// TIA Portal V20 export
// export: Created 2025-12-01T14:56:34.8716322Z, ExportSetting None, DisplayName Totally Integrated Automation Portal, DisplayVersion V20 Update 3, DisplayName TIA Portal Openness, DisplayVersion V20 Update 3, DisplayName TIA Portal Version Control Interface, DisplayVersion V20 Update 3, DisplayName STEP 7 Professional, DisplayVersion V20 Update 3, DisplayName STEP 7 Safety, DisplayVersion V20 Update 2, DisplayName WinCC Basic/Comfort/Advanced, DisplayVersion V20 Update 3, DisplayName WinCC Professional, DisplayVersion V20 Update 3, DisplayName WinCC Unified, DisplayVersion V20 Update 3
FUNCTION_BLOCK "FB464_CRTL_TR_TP_E124_S34_Pres"   // FB464, LAD
TITLE = bimba y lola
{ S7_Optimized_Access := 'FALSE' }
AUTHOR : TLigero
NAME : 20180827
VERSION : 3.0
// pendiente de simular
// stored: AutoNumber false, SetENOAutomatically false
   VAR_INPUT
      Mesa : UInt;   // Número de mesa
      En_Tension : Bool;
      pHsMx : Bool;   // pHs de presencia de la Mesa
      TP1_Up : Bool;   // TP1 Arriba. E1 >> S3. si no hay tope poner ON
      TP1_Down : Bool;   // TP1 Abajo. E1 >> S3. si no hay tope poner ON
      PosTR_E1 : Bool;   // Posicion del TR en E1E3
      PosTR_E2 { ExternalVisible := 'False'} : Bool;   // Posicion del TR en E2E4
      Termico_13 : Bool;   // Proteccion del Tx en E1E3
      Termico_24 : Bool;   // Proteccion del Tx en E2E4
      Avance_13 : Bool;   // Avance del Tx en E1E3
      Avance_24 : Bool;   // Avance del Tx en E2E4
      PTF_Sal_M3 : Bool;   // S3 >> Mesa Siguiente PTF
      NXT_Avance_S3 : Bool;   // S3 >> Mesa Siguiente PTF
      PTF_Sal_M4 : Bool;   // S4 >> Mesa Siguiente PTF
      NXT_Avance_S4 : Bool;   // S4 >> Mesa Siguiente PTF
      Mx_Bloq_Activo : Bool;   // Bloqueo Activo de la Mesa
      Mx_FlujoPrin_S4 : Bool;   // El flujo principal es Saliendo por S4
      F_EnvMens_Mx : Bool;   // Fin de Envio de Mensaje
      AVTF_Ent_M1 : Bool;   // E1 >> Mesa Anterior AVTF
      AVTF_Ent_M2 : Bool;   // E2 >> Mesa Anterior AVTF
      AVTF_Ent_M4 : Bool;   // E4 >> Mesa Anterior AVTF
      Num_Cruce : UInt;   // Número de cruce.
      DB_FIFO_Cruce : UInt := 213;   // DB de la FIFO de ordenes del cruce
      Long_FIFO_Cruce : UInt := 1;   // Longitut de la FIFO de ordenes del cruce
      ValorOrden_S4 : Word := 16#81;   // Con que orden entra por S4
      MesaS3 : UInt;   // Número de mesa por S3
      MesaS4 : UInt;   // Número de mesa por S4
      V_CNT_pHsMx_E1 : UDInt := 500;   // Valor de presencia por E1 en ms
      V_CNT_pHsMx_E2 : UDInt := 500;   // Valor de presencia por E2 en ms
      V_CNT_pHsMx_E4 : UDInt := 500;   // Valor de presencia por E4 en ms
      V_CNT_ApHsMx_S3 : UDInt := 500;   // Valor de Ausencia por S3 en ms
      V_CNT_ApHsMx_S4 : UDInt := 500;   // Valor de Ausencia por S4 en ms
      V_TOut_Tx_Mx : UDInt := 3000;   // TimeOut de Atasco en ms
      V_TOut_TP : UDInt := 2000;   // TimeOut de Tope en ms
      V_TOut_TR : UDInt := 2000;   // TimeOut de Transfer en ms
      V_Paro : UDInt := 5000;   // tiempo que avanza el transportador sin aviso hasta que se para (ms)
      V_Vaciado : UDInt := 5000;   // Valor de vaciado en ms
   END_VAR
   VAR_OUTPUT
      P_EnvMens_PMx : Bool;   // Permiso de Enviar Mensaje de Presencia
      Etiqueta_Jdt : UDInt;   // Etiqueta que ha sido leida
      Orden_Ejecutada_Jdt : UInt;   // Orden que se ha ejecutado
      PTF_Ent_M1 : Bool;   // E1 >> Mesa Anterior PTF
      PTF_Ent_M2 : Bool;   // E2 >> Mesa Anterior PTF
      PTF_Ent_M4 : Bool;
      AVTF_Sal_M3 : Bool;   // S3 >> Mesa Siguiente AVTF
      NXT_Descarga_Act_S3 : Bool;   // S3 >> Mesa Siguiente descarga activa
      AVTF_Sal_M4 : Bool;   // S4 >> Mesa Siguiente AVTF
      NXT_Descarga_Act_S4 : Bool;   // S4 >> Mesa Siguiente descarga activa
   END_VAR
   VAR
      T1_ET00 : Bool;
      T1_ET01 : Bool;
      T1_ET02 : Bool;
      T1_ET03 : Bool;
      T1_ET10 : Bool;
      T1_ET11 : Bool;
      T1_ET20 : Bool;
      T1_ET21 : Bool;
      T1_ET50 : Bool;
      T1_ET60 : Bool;
      T1_ET110 : Bool;
      T1_ET111 : Bool;
      T1_ET112 : Bool;
      FIFO_OK : Bool;
      TRANS_OK : Bool;
      O_Bloqueo : Bool;
      Selec_M2_Entrada : Bool;
      Selec_M4_Entrada : Bool;
      Inv_Avance : Bool;
      maux_fp_disparo_e1 : Bool;
      maux_fp_disparo_e2 : Bool;
      Err_Detec_PHS : Bool;
      tim_vaciado_Q : Bool;
      Tim_paro_Q : Bool;
      TMP_Tout_Tp_Q : Bool;
      Tmp_tout_tr_Q : Bool;
      TMP_Atasco_Q : Bool;
      FN_ET02 : Bool;
      TMP_pHs_E1 : UDInt;
      CNT_pHs_E2 : UDInt;
      CNT_pHs_E4 : UDInt;
      TMP_Aus_S3 : UDInt;
      TMP_Aus_S4 : UDInt;
      TIM_Vaciado : UDInt;
      TMP_Paro : UDInt;
      TMP_Tout_Tp : UDInt;
      TMP_Tout_Tr : UDInt;
      TMP_atasco : UDInt;
      TMP_En_Tension : UDInt;
      Datos_Scanner { S7_SetPoint := 'True'} : "ROUT_Orden_Fifo_Scanner";
   END_VAR
   VAR_TEMP
      EstadoZona : "EstadoZona";   // Estado de Zona de la Mesa
      EstadoVI : "EstadosMesa";   // Estado del Vehiculo Inteliguente de la Mesa
      ConfigFB : "UDT_ConfigFB";   // Configuracion de la FB de la Mesa
      MA_SubirTP : Bool;
      O_Sal_S3 : Bool;
      O_Sal_S4 : Bool;
      O_Vaciar : Bool;
      Moti_ERRO : Bool;
      Moti_NENC : Bool;
      Moti_NORM : Bool;
      Moti_INIC : Bool;
      tmp_pHs_E1_Q : Bool;
      tmp_pHs_E2_Q : Bool;
      tmp_pHs_E4_Q : Bool;
      tmp_Aus_S4_Q : Bool;
      tmp_pHs_S3_Q : Bool;
      ok_tension : Bool;
      Aux_W_Moti : Word;
      INT_ORDEN : UInt;
      Aux_W_Orden : Word;
      I_Ord_Filtrada : UInt;
      I_V_Ord_S4 : UInt;
   END_VAR
   VAR_TEMP   // added for the SCL form of the ladder/FBD networks
      _w1 : Bool;
      _w2 : Bool;
      _w3 : Bool;
      _w4 : Bool;
      _w5 : Bool;
      _w6 : Bool;
   END_VAR
BEGIN

REGION Network 1: INICIALIZAR - Recoger las Variables de Estado de la Mesa
   // Se recoge - Estado_CBx
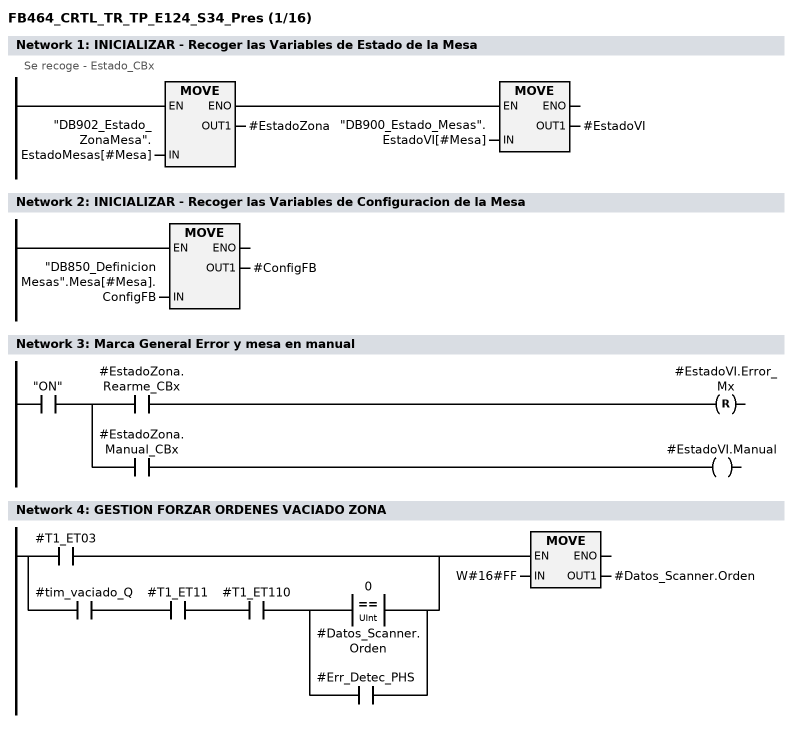
   RUNG wire#powerrail
      Move(in := "DB902_Estado_ZonaMesa".EstadoMesas[#Mesa], out1 => #EstadoZona)
      Move(in := "DB900_Estado_Mesas".EstadoVI[#Mesa], out1 => #EstadoVI)
   END_RUNG
   // the same network as SCL:
   #EstadoZona := "DB902_Estado_ZonaMesa".EstadoMesas[#Mesa];
   #EstadoVI := "DB900_Estado_Mesas".EstadoVI[#Mesa];
END_REGION

REGION Network 2: INICIALIZAR - Recoger las Variables de Configuracion de la Mesa
   RUNG wire#powerrail
      Move(in := "DB850_DefinicionMesas".Mesa[#Mesa].ConfigFB, out1 => #ConfigFB)
   END_RUNG
   // the same network as SCL:
   #ConfigFB := "DB850_DefinicionMesas".Mesa[#Mesa].ConfigFB;
END_REGION

REGION Network 3: Marca General Error y mesa en manual
   RUNG wire#powerrail
      Contact( "ON" )
      wire#w1
      Contact( #EstadoZona.Rearme_CBx )
      R_Coil( #EstadoVI.Error_Mx )
   END_RUNG
   RUNG wire#w1
      Contact( #EstadoZona.Manual_CBx )
      Coil( #EstadoVI.Manual )
   END_RUNG
   // the same network as SCL:
   IF "ON" AND #EstadoZona.Rearme_CBx THEN #EstadoVI.Error_Mx := FALSE; END_IF;
   #EstadoVI.Manual := "ON" AND #EstadoZona.Manual_CBx;
END_REGION

REGION Network 4: GESTION FORZAR ORDENES VACIADO ZONA
   RUNG wire#powerrail
      Contact( #T1_ET03 )
      wire#w1
      { S7_GenerateENO := "TRUE" } Move(in := W#16#FF, out1 => #Datos_Scanner.Orden)
   END_RUNG
   RUNG wire#powerrail
      Contact( #tim_vaciado_Q )
      Contact( #T1_ET11 )
      Contact( #T1_ET110 )
      wire#w2
      { S7_Templates := "SrcType := UInt" } EQ_Contact(in1 := 0, in2 := #Datos_Scanner.Orden)
   END_RUNG wire#w1
   RUNG wire#w2
      Contact( #Err_Detec_PHS )
   END_RUNG wire#w1
   // the same network as SCL:
   IF #T1_ET03 OR (#tim_vaciado_Q AND #T1_ET11 AND #T1_ET110 AND ((0 = #Datos_Scanner.Orden) OR #Err_Detec_PHS)) THEN
       #Datos_Scanner.Orden := W#16#FF;
   END_IF;
END_REGION

REGION Network 5: Extraer orden
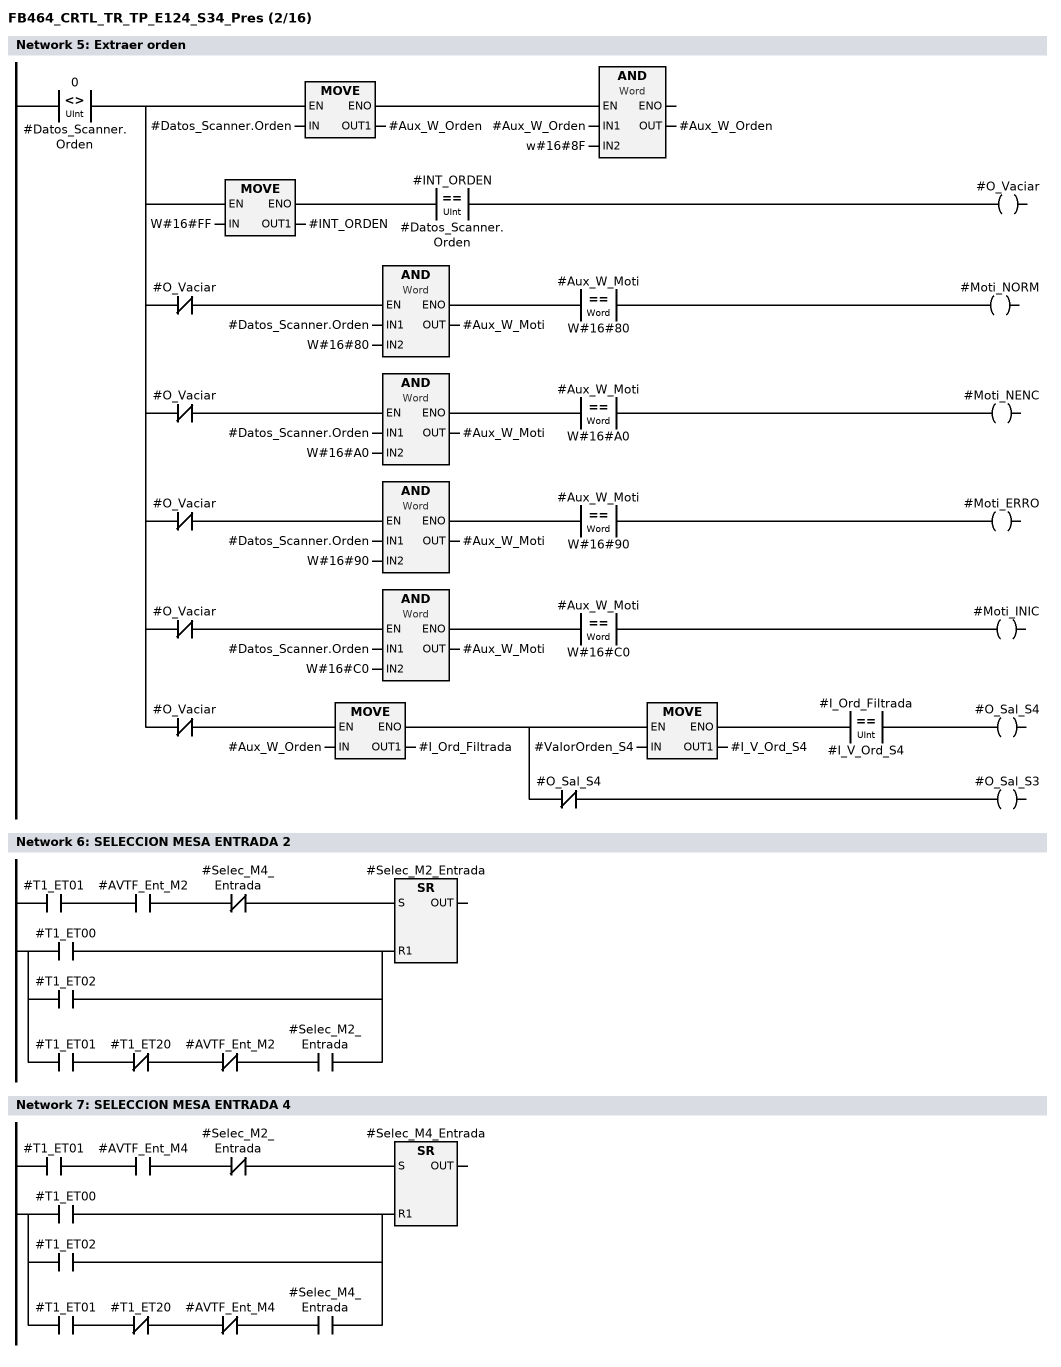
   RUNG wire#powerrail
      { S7_Templates := "SrcType := UInt" } NE_Contact(in1 := 0, in2 := #Datos_Scanner.Orden)
      wire#w1
      { S7_GenerateENO := "TRUE" } Move(in := #Datos_Scanner.Orden, out1 => #Aux_W_Orden)
      { S7_Templates := "SrcType := Word"; S7_GenerateENO := "TRUE" } And(in1 := #Aux_W_Orden, in2 := w#16#8F, out => #Aux_W_Orden)
   END_RUNG
   RUNG wire#w1
      { S7_GenerateENO := "TRUE" } Move(in := W#16#FF, out1 => #INT_ORDEN)
      { S7_Templates := "SrcType := UInt" } EQ_Contact(in1 := #INT_ORDEN, in2 := #Datos_Scanner.Orden)
      Coil( #O_Vaciar )
   END_RUNG
   RUNG wire#w1
      I_Contact( #O_Vaciar )
      { S7_Templates := "SrcType := Word"; S7_GenerateENO := "TRUE" } And(in1 := #Datos_Scanner.Orden, in2 := W#16#80, out => #Aux_W_Moti)
      { S7_Templates := "SrcType := Word" } EQ_Contact(in1 := #Aux_W_Moti, in2 := W#16#80)
      Coil( #Moti_NORM )
   END_RUNG
   RUNG wire#w1
      I_Contact( #O_Vaciar )
      { S7_Templates := "SrcType := Word"; S7_GenerateENO := "TRUE" } And(in1 := #Datos_Scanner.Orden, in2 := W#16#A0, out => #Aux_W_Moti)
      { S7_Templates := "SrcType := Word" } EQ_Contact(in1 := #Aux_W_Moti, in2 := W#16#A0)
      Coil( #Moti_NENC )
   END_RUNG
   RUNG wire#w1
      I_Contact( #O_Vaciar )
      { S7_Templates := "SrcType := Word"; S7_GenerateENO := "TRUE" } And(in1 := #Datos_Scanner.Orden, in2 := W#16#90, out => #Aux_W_Moti)
      { S7_Templates := "SrcType := Word" } EQ_Contact(in1 := #Aux_W_Moti, in2 := W#16#90)
      Coil( #Moti_ERRO )
   END_RUNG
   RUNG wire#w1
      I_Contact( #O_Vaciar )
      { S7_Templates := "SrcType := Word"; S7_GenerateENO := "TRUE" } And(in1 := #Datos_Scanner.Orden, in2 := W#16#C0, out => #Aux_W_Moti)
      { S7_Templates := "SrcType := Word" } EQ_Contact(in1 := #Aux_W_Moti, in2 := W#16#C0)
      Coil( #Moti_INIC )
   END_RUNG
   RUNG wire#w1
      I_Contact( #O_Vaciar )
      { S7_GenerateENO := "TRUE" } Move(in := #Aux_W_Orden, out1 => #I_Ord_Filtrada)
      wire#w2
      { S7_GenerateENO := "TRUE" } Move(in := #ValorOrden_S4, out1 => #I_V_Ord_S4)
      { S7_Templates := "SrcType := UInt" } EQ_Contact(in1 := #I_Ord_Filtrada, in2 := #I_V_Ord_S4)
      Coil( #O_Sal_S4 )
   END_RUNG
   RUNG wire#w2
      I_Contact( #O_Sal_S4 )
      Coil( #O_Sal_S3 )
   END_RUNG
   // the same network as SCL:
   // ENO of a box is taken as its EN; it also drops when the box reports an error
   #_w1 := 0 <> #Datos_Scanner.Orden;
   IF #_w1 THEN
       #Aux_W_Orden := #Datos_Scanner.Orden;
       #Aux_W_Orden := #Aux_W_Orden AND w#16#8F;
       #INT_ORDEN := W#16#FF;
   END_IF;
   #O_Vaciar := #_w1 AND (#INT_ORDEN = #Datos_Scanner.Orden);
   #_w2 := #_w1 AND NOT #O_Vaciar;
   IF #_w2 THEN #Aux_W_Moti := #Datos_Scanner.Orden AND W#16#80; END_IF;
   #Moti_NORM := #_w2 AND (#Aux_W_Moti = W#16#80);
   #_w3 := #_w1 AND NOT #O_Vaciar;
   IF #_w3 THEN #Aux_W_Moti := #Datos_Scanner.Orden AND W#16#A0; END_IF;
   #Moti_NENC := #_w3 AND (#Aux_W_Moti = W#16#A0);
   #_w4 := #_w1 AND NOT #O_Vaciar;
   IF #_w4 THEN #Aux_W_Moti := #Datos_Scanner.Orden AND W#16#90; END_IF;
   #Moti_ERRO := #_w4 AND (#Aux_W_Moti = W#16#90);
   #_w5 := #_w1 AND NOT #O_Vaciar;
   IF #_w5 THEN #Aux_W_Moti := #Datos_Scanner.Orden AND W#16#C0; END_IF;
   #Moti_INIC := #_w5 AND (#Aux_W_Moti = W#16#C0);
   #_w6 := #_w1 AND NOT #O_Vaciar;
   IF #_w6 THEN
       #I_Ord_Filtrada := #Aux_W_Orden;
       #I_V_Ord_S4 := #ValorOrden_S4;
   END_IF;
   #O_Sal_S4 := #_w6 AND (#I_Ord_Filtrada = #I_V_Ord_S4);
   #O_Sal_S3 := #_w6 AND NOT #O_Sal_S4;
END_REGION

REGION Network 6: SELECCION MESA ENTRADA 2
   RUNG wire#powerrail
      Contact( #T1_ET01 )
      Contact( #AVTF_Ent_M2 )
      I_Contact( #Selec_M4_Entrada )
      S_SR(operand := #Selec_M2_Entrada, r1 := wire#w1)
   END_RUNG
   RUNG wire#powerrail
      Contact( #T1_ET00 )
   END_RUNG wire#w1
   RUNG wire#powerrail
      Contact( #T1_ET02 )
   END_RUNG wire#w1
   RUNG wire#powerrail
      Contact( #T1_ET01 )
      I_Contact( #T1_ET20 )
      I_Contact( #AVTF_Ent_M2 )
      Contact( #Selec_M2_Entrada )
   END_RUNG wire#w1
   // the same network as SCL:
   #_w1 := #T1_ET00 OR #T1_ET02 OR (#T1_ET01 AND NOT #T1_ET20 AND NOT #AVTF_Ent_M2 AND #Selec_M2_Entrada);
   IF #T1_ET01 AND #AVTF_Ent_M2 AND NOT #Selec_M4_Entrada THEN
       #Selec_M2_Entrada := TRUE;   // SR flip-flop
   END_IF;
   IF #_w1 THEN #Selec_M2_Entrada := FALSE; END_IF;
END_REGION

REGION Network 7: SELECCION MESA ENTRADA 4
   RUNG wire#powerrail
      Contact( #T1_ET01 )
      Contact( #AVTF_Ent_M4 )
      I_Contact( #Selec_M2_Entrada )
      S_SR(operand := #Selec_M4_Entrada, r1 := wire#w1)
   END_RUNG
   RUNG wire#powerrail
      Contact( #T1_ET00 )
   END_RUNG wire#w1
   RUNG wire#powerrail
      Contact( #T1_ET02 )
   END_RUNG wire#w1
   RUNG wire#powerrail
      Contact( #T1_ET01 )
      I_Contact( #T1_ET20 )
      I_Contact( #AVTF_Ent_M4 )
      Contact( #Selec_M4_Entrada )
   END_RUNG wire#w1
   // the same network as SCL:
   #_w1 := #T1_ET00 OR #T1_ET02 OR (#T1_ET01 AND NOT #T1_ET20 AND NOT #AVTF_Ent_M4 AND #Selec_M4_Entrada);
   IF #T1_ET01 AND #AVTF_Ent_M4 AND NOT #Selec_M2_Entrada THEN
       #Selec_M4_Entrada := TRUE;   // SR flip-flop
   END_IF;
   IF #_w1 THEN #Selec_M4_Entrada := FALSE; END_IF;
END_REGION

REGION Network 8: #T1_ET60. SALIR POR S4
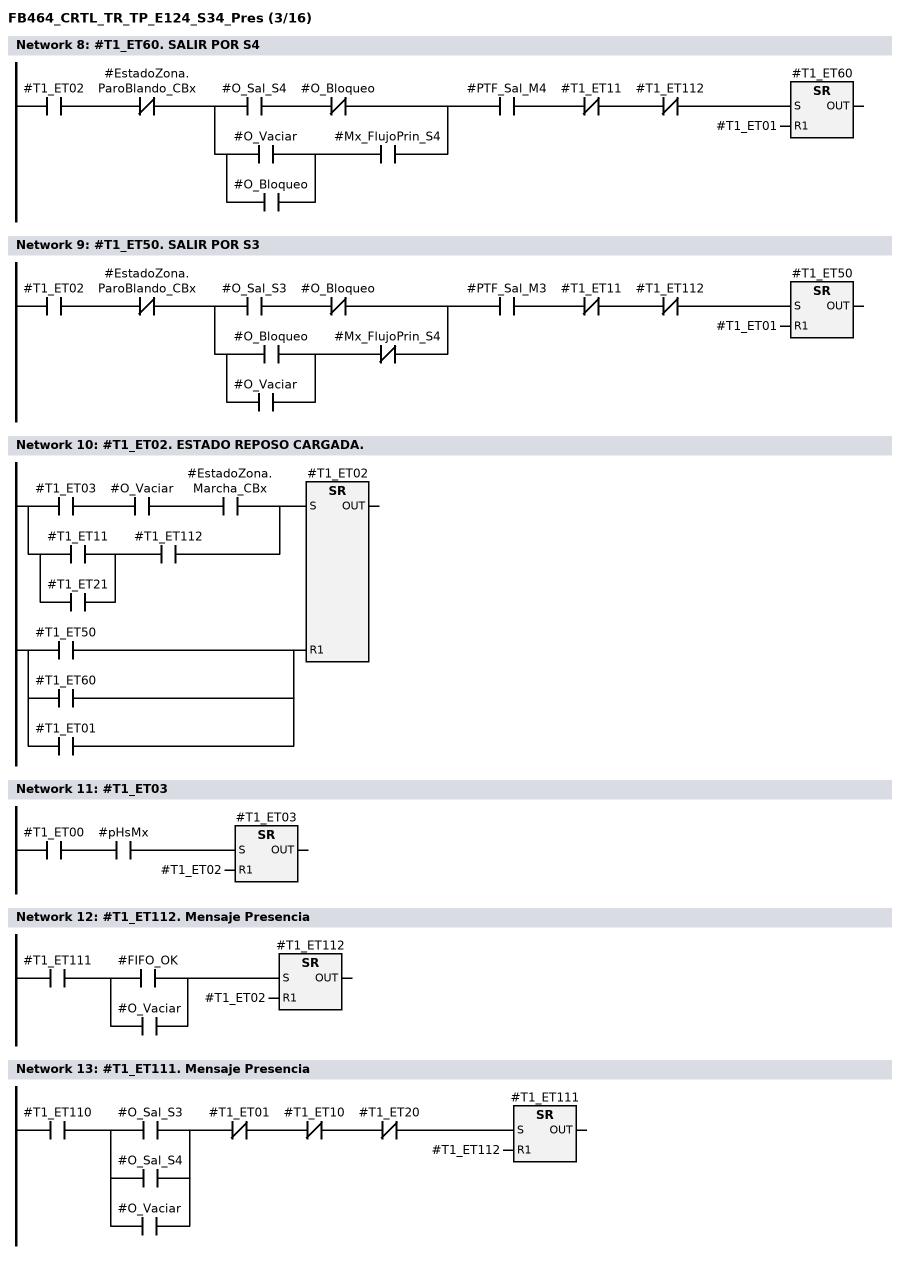
   RUNG wire#powerrail
      Contact( #T1_ET02 )
      I_Contact( #EstadoZona.ParoBlando_CBx )
      wire#w1
      Contact( #O_Sal_S4 )
      I_Contact( #O_Bloqueo )
      wire#w2
      Contact( #PTF_Sal_M4 )
      I_Contact( #T1_ET11 )
      I_Contact( #T1_ET112 )
      S_SR(operand := #T1_ET60, r1 := #T1_ET01)
   END_RUNG
   RUNG wire#w1
      Contact( #O_Vaciar )
      wire#w3
      Contact( #Mx_FlujoPrin_S4 )
   END_RUNG wire#w2
   RUNG wire#w1
      Contact( #O_Bloqueo )
   END_RUNG wire#w3
   // the same network as SCL:
   IF #T1_ET02 AND NOT #EstadoZona.ParoBlando_CBx AND ((#O_Sal_S4 AND NOT #O_Bloqueo) OR ((#O_Vaciar OR #O_Bloqueo) AND #Mx_FlujoPrin_S4)) AND #PTF_Sal_M4 AND NOT #T1_ET11 AND NOT #T1_ET112 THEN
       #T1_ET60 := TRUE;   // SR flip-flop
   END_IF;
   IF #T1_ET01 THEN #T1_ET60 := FALSE; END_IF;
END_REGION

REGION Network 9: #T1_ET50. SALIR POR S3
   RUNG wire#powerrail
      Contact( #T1_ET02 )
      I_Contact( #EstadoZona.ParoBlando_CBx )
      wire#w1
      Contact( #O_Sal_S3 )
      I_Contact( #O_Bloqueo )
      wire#w2
      Contact( #PTF_Sal_M3 )
      I_Contact( #T1_ET11 )
      I_Contact( #T1_ET112 )
      S_SR(operand := #T1_ET50, r1 := #T1_ET01)
   END_RUNG
   RUNG wire#w1
      Contact( #O_Bloqueo )
      wire#w3
      I_Contact( #Mx_FlujoPrin_S4 )
   END_RUNG wire#w2
   RUNG wire#w1
      Contact( #O_Vaciar )
   END_RUNG wire#w3
   // the same network as SCL:
   IF #T1_ET02 AND NOT #EstadoZona.ParoBlando_CBx AND ((#O_Sal_S3 AND NOT #O_Bloqueo) OR ((#O_Bloqueo OR #O_Vaciar) AND NOT #Mx_FlujoPrin_S4)) AND #PTF_Sal_M3 AND NOT #T1_ET11 AND NOT #T1_ET112 THEN
       #T1_ET50 := TRUE;   // SR flip-flop
   END_IF;
   IF #T1_ET01 THEN #T1_ET50 := FALSE; END_IF;
END_REGION

REGION Network 10: #T1_ET02. ESTADO REPOSO CARGADA.
   RUNG wire#powerrail
      Contact( #T1_ET03 )
      Contact( #O_Vaciar )
      Contact( #EstadoZona.Marcha_CBx )
      wire#w1
      S_SR(operand := #T1_ET02, r1 := wire#w3)
   END_RUNG
   RUNG wire#powerrail
      Contact( #T1_ET11 )
      wire#w2
      Contact( #T1_ET112 )
   END_RUNG wire#w1
   RUNG wire#powerrail
      Contact( #T1_ET21 )
   END_RUNG wire#w2
   RUNG wire#powerrail
      Contact( #T1_ET50 )
   END_RUNG wire#w3
   RUNG wire#powerrail
      Contact( #T1_ET60 )
   END_RUNG wire#w3
   RUNG wire#powerrail
      Contact( #T1_ET01 )
   END_RUNG wire#w3
   // the same network as SCL:
   IF (#T1_ET03 AND #O_Vaciar AND #EstadoZona.Marcha_CBx) OR ((#T1_ET11 OR #T1_ET21) AND #T1_ET112) THEN
       #T1_ET02 := TRUE;   // SR flip-flop
   END_IF;
   IF #T1_ET50 OR #T1_ET60 OR #T1_ET01 THEN #T1_ET02 := FALSE; END_IF;
END_REGION

REGION Network 11: #T1_ET03
   RUNG wire#powerrail
      Contact( #T1_ET00 )
      Contact( #pHsMx )
      S_SR(operand := #T1_ET03, r1 := #T1_ET02)
   END_RUNG
   // the same network as SCL:
   IF #T1_ET00 AND #pHsMx THEN
       #T1_ET03 := TRUE;   // SR flip-flop
   END_IF;
   IF #T1_ET02 THEN #T1_ET03 := FALSE; END_IF;
END_REGION

REGION Network 12: #T1_ET112. Mensaje Presencia
   RUNG wire#powerrail
      Contact( #T1_ET111 )
      wire#w1
      Contact( #FIFO_OK )
      wire#w2
      S_SR(operand := #T1_ET112, r1 := #T1_ET02)
   END_RUNG
   RUNG wire#w1
      Contact( #O_Vaciar )
   END_RUNG wire#w2
   // the same network as SCL:
   IF #T1_ET111 AND (#FIFO_OK OR #O_Vaciar) THEN
       #T1_ET112 := TRUE;   // SR flip-flop
   END_IF;
   IF #T1_ET02 THEN #T1_ET112 := FALSE; END_IF;
END_REGION

REGION Network 13: #T1_ET111. Mensaje Presencia
   RUNG wire#powerrail
      Contact( #T1_ET110 )
      wire#w1
      Contact( #O_Sal_S3 )
      wire#w2
      I_Contact( #T1_ET01 )
      I_Contact( #T1_ET10 )
      I_Contact( #T1_ET20 )
      S_SR(operand := #T1_ET111, r1 := #T1_ET112)
   END_RUNG
   RUNG wire#w1
      Contact( #O_Sal_S4 )
   END_RUNG wire#w2
   RUNG wire#w1
      Contact( #O_Vaciar )
   END_RUNG wire#w2
   // the same network as SCL:
   IF #T1_ET110 AND (#O_Sal_S3 OR #O_Sal_S4 OR #O_Vaciar) AND NOT #T1_ET01 AND NOT #T1_ET10 AND NOT #T1_ET20 THEN
       #T1_ET111 := TRUE;   // SR flip-flop
   END_IF;
   IF #T1_ET112 THEN #T1_ET111 := FALSE; END_IF;
END_REGION

REGION Network 14: #T1_ET110
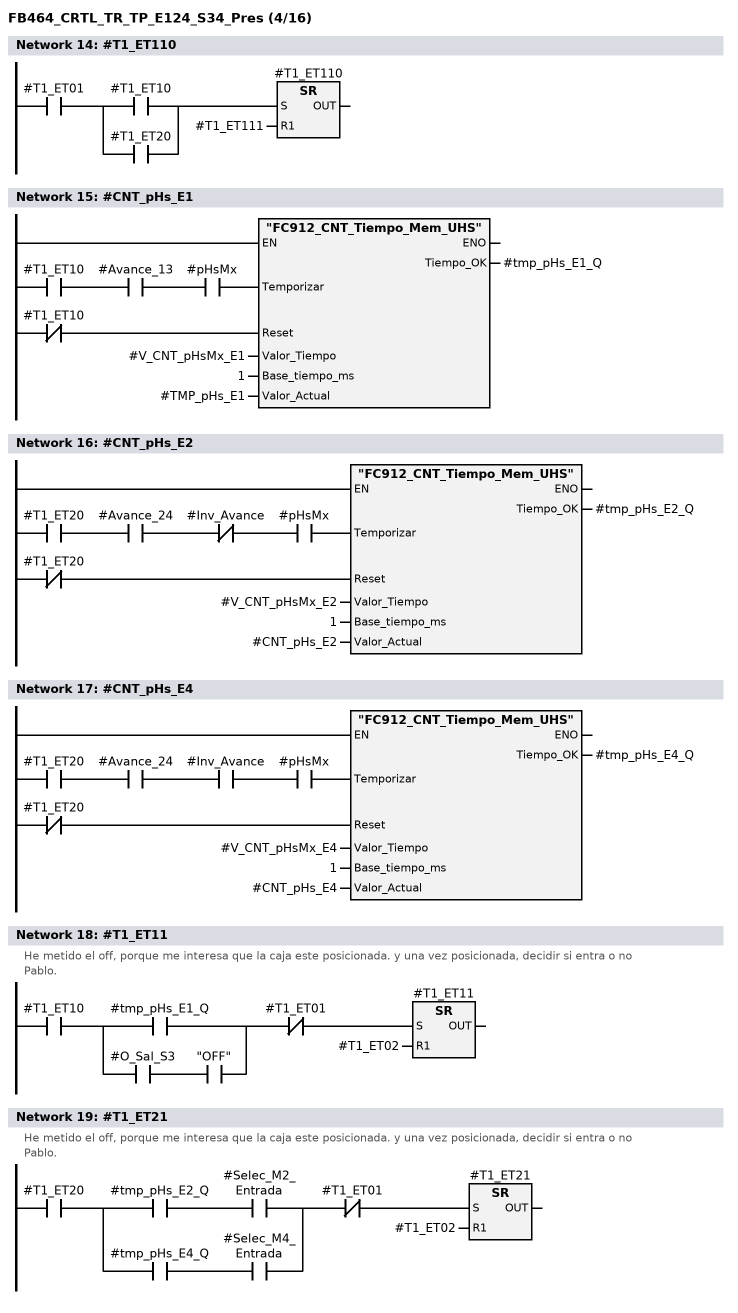
   RUNG wire#powerrail
      Contact( #T1_ET01 )
      wire#w1
      Contact( #T1_ET10 )
      wire#w2
      S_SR(operand := #T1_ET110, r1 := #T1_ET111)
   END_RUNG
   RUNG wire#w1
      Contact( #T1_ET20 )
   END_RUNG wire#w2
   // the same network as SCL:
   IF #T1_ET01 AND (#T1_ET10 OR #T1_ET20) THEN
       #T1_ET110 := TRUE;   // SR flip-flop
   END_IF;
   IF #T1_ET111 THEN #T1_ET110 := FALSE; END_IF;
END_REGION

REGION Network 15: #CNT_pHs_E1
   RUNG wire#powerrail
      "FC912_CNT_Tiempo_Mem_UHS"(Temporizar := wire#w1, Reset := wire#w2, Valor_Tiempo := #V_CNT_pHsMx_E1, Base_tiempo_ms := 1, Valor_Actual := #TMP_pHs_E1, Tiempo_OK => #tmp_pHs_E1_Q)
   END_RUNG
   RUNG wire#powerrail
      Contact( #T1_ET10 )
      Contact( #Avance_13 )
      Contact( #pHsMx )
   END_RUNG wire#w1
   RUNG wire#powerrail
      I_Contact( #T1_ET10 )
   END_RUNG wire#w2
   // the same network as SCL:
   "FC912_CNT_Tiempo_Mem_UHS"(Temporizar := #T1_ET10 AND #Avance_13 AND #pHsMx,
                           Reset := NOT #T1_ET10,
                           Valor_Tiempo := #V_CNT_pHsMx_E1,
                           Base_tiempo_ms := 1,
                           Valor_Actual := #TMP_pHs_E1,
                           Tiempo_OK => #tmp_pHs_E1_Q);
END_REGION

REGION Network 16: #CNT_pHs_E2
   RUNG wire#powerrail
      "FC912_CNT_Tiempo_Mem_UHS"(Temporizar := wire#w1, Reset := wire#w2, Valor_Tiempo := #V_CNT_pHsMx_E2, Base_tiempo_ms := 1, Valor_Actual := #CNT_pHs_E2, Tiempo_OK => #tmp_pHs_E2_Q)
   END_RUNG
   RUNG wire#powerrail
      Contact( #T1_ET20 )
      Contact( #Avance_24 )
      I_Contact( #Inv_Avance )
      Contact( #pHsMx )
   END_RUNG wire#w1
   RUNG wire#powerrail
      I_Contact( #T1_ET20 )
   END_RUNG wire#w2
   // the same network as SCL:
   "FC912_CNT_Tiempo_Mem_UHS"(Temporizar := #T1_ET20 AND #Avance_24 AND NOT #Inv_Avance AND #pHsMx,
                           Reset := NOT #T1_ET20,
                           Valor_Tiempo := #V_CNT_pHsMx_E2,
                           Base_tiempo_ms := 1,
                           Valor_Actual := #CNT_pHs_E2,
                           Tiempo_OK => #tmp_pHs_E2_Q);
END_REGION

REGION Network 17: #CNT_pHs_E4
   RUNG wire#powerrail
      "FC912_CNT_Tiempo_Mem_UHS"(Temporizar := wire#w1, Reset := wire#w2, Valor_Tiempo := #V_CNT_pHsMx_E4, Base_tiempo_ms := 1, Valor_Actual := #CNT_pHs_E4, Tiempo_OK => #tmp_pHs_E4_Q)
   END_RUNG
   RUNG wire#powerrail
      Contact( #T1_ET20 )
      Contact( #Avance_24 )
      Contact( #Inv_Avance )
      Contact( #pHsMx )
   END_RUNG wire#w1
   RUNG wire#powerrail
      I_Contact( #T1_ET20 )
   END_RUNG wire#w2
   // the same network as SCL:
   "FC912_CNT_Tiempo_Mem_UHS"(Temporizar := #T1_ET20 AND #Avance_24 AND #Inv_Avance AND #pHsMx,
                           Reset := NOT #T1_ET20,
                           Valor_Tiempo := #V_CNT_pHsMx_E4,
                           Base_tiempo_ms := 1,
                           Valor_Actual := #CNT_pHs_E4,
                           Tiempo_OK => #tmp_pHs_E4_Q);
END_REGION

REGION Network 18: #T1_ET11
   // He metido el off, porque me interesa que la caja este posicionada. y una vez posicionada, decidir si entra o no
   // Pablo.
   RUNG wire#powerrail
      Contact( #T1_ET10 )
      wire#w1
      Contact( #tmp_pHs_E1_Q )
      wire#w2
      I_Contact( #T1_ET01 )
      S_SR(operand := #T1_ET11, r1 := #T1_ET02)
   END_RUNG
   RUNG wire#w1
      Contact( #O_Sal_S3 )
      Contact( "OFF" )
   END_RUNG wire#w2
   // the same network as SCL:
   IF #T1_ET10 AND (#tmp_pHs_E1_Q OR (#O_Sal_S3 AND "OFF")) AND NOT #T1_ET01 THEN
       #T1_ET11 := TRUE;   // SR flip-flop
   END_IF;
   IF #T1_ET02 THEN #T1_ET11 := FALSE; END_IF;
END_REGION

REGION Network 19: #T1_ET21
   // He metido el off, porque me interesa que la caja este posicionada. y una vez posicionada, decidir si entra o no
   // Pablo.
   RUNG wire#powerrail
      Contact( #T1_ET20 )
      wire#w1
      Contact( #tmp_pHs_E2_Q )
      Contact( #Selec_M2_Entrada )
      wire#w2
      I_Contact( #T1_ET01 )
      S_SR(operand := #T1_ET21, r1 := #T1_ET02)
   END_RUNG
   RUNG wire#w1
      Contact( #tmp_pHs_E4_Q )
      Contact( #Selec_M4_Entrada )
   END_RUNG wire#w2
   // the same network as SCL:
   IF #T1_ET20 AND ((#tmp_pHs_E2_Q AND #Selec_M2_Entrada) OR (#tmp_pHs_E4_Q AND #Selec_M4_Entrada)) AND NOT #T1_ET01 THEN
       #T1_ET21 := TRUE;   // SR flip-flop
   END_IF;
   IF #T1_ET02 THEN #T1_ET21 := FALSE; END_IF;
END_REGION

REGION Network 20: #T1_ET10.
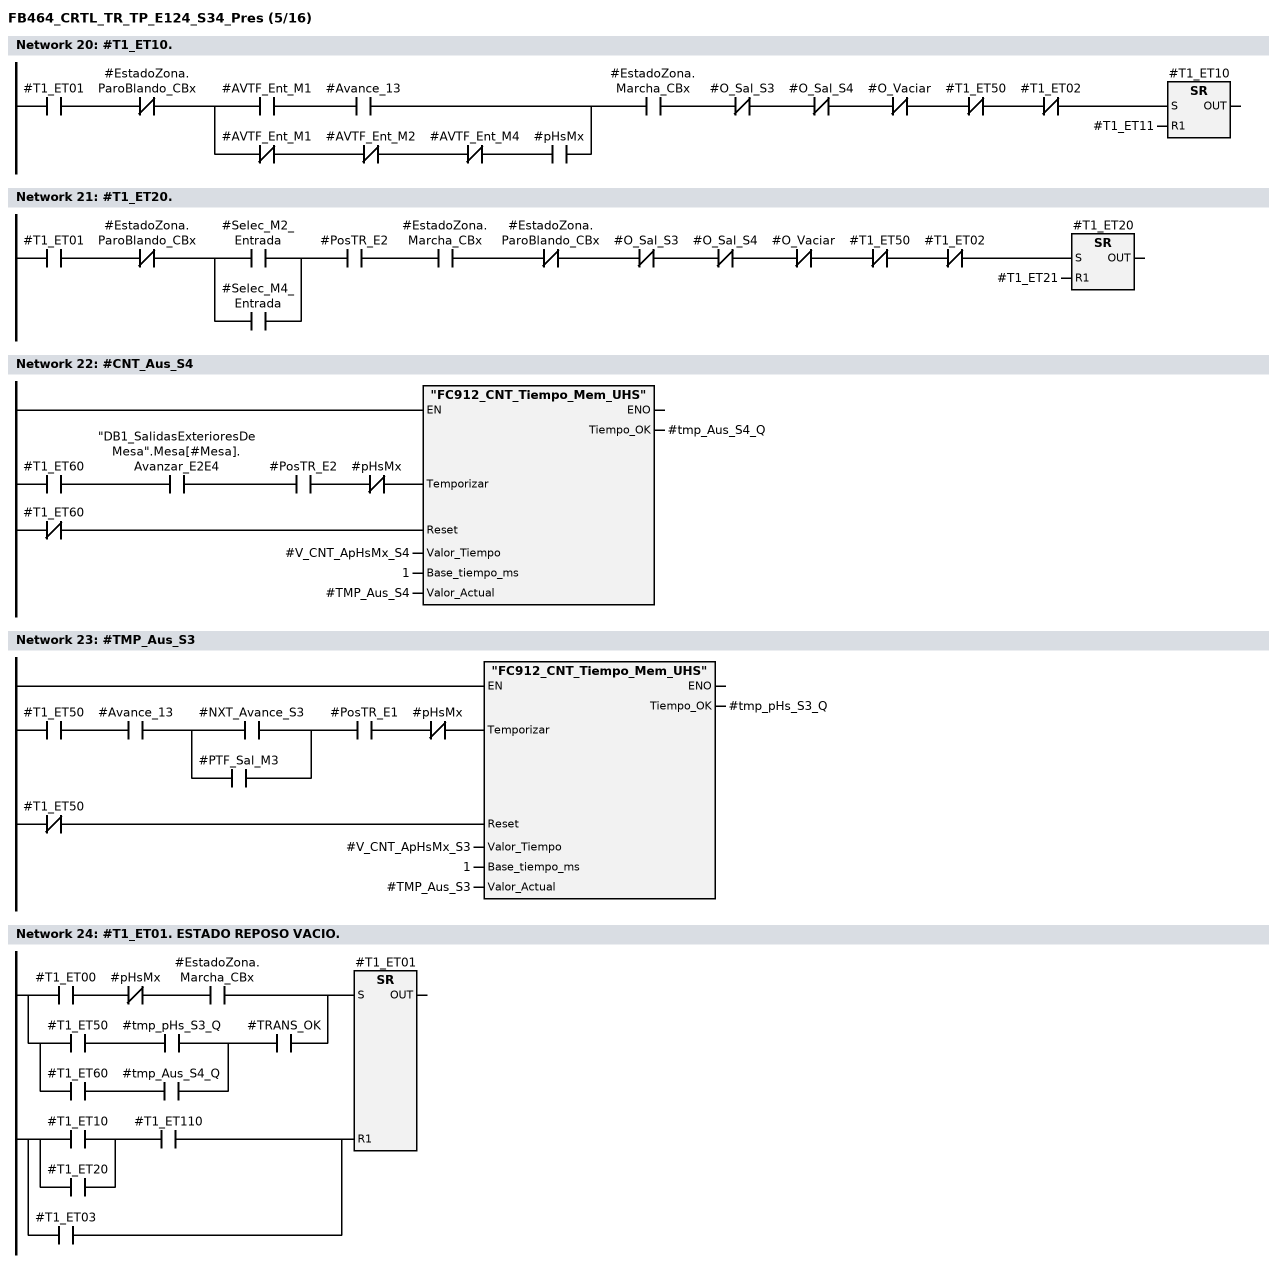
   RUNG wire#powerrail
      Contact( #T1_ET01 )
      I_Contact( #EstadoZona.ParoBlando_CBx )
      wire#w1
      Contact( #AVTF_Ent_M1 )
      Contact( #Avance_13 )
      wire#w2
      Contact( #EstadoZona.Marcha_CBx )
      I_Contact( #O_Sal_S3 )
      I_Contact( #O_Sal_S4 )
      I_Contact( #O_Vaciar )
      I_Contact( #T1_ET50 )
      I_Contact( #T1_ET02 )
      S_SR(operand := #T1_ET10, r1 := #T1_ET11)
   END_RUNG
   RUNG wire#w1
      I_Contact( #AVTF_Ent_M1 )
      I_Contact( #AVTF_Ent_M2 )
      I_Contact( #AVTF_Ent_M4 )
      Contact( #pHsMx )
   END_RUNG wire#w2
   // the same network as SCL:
   IF #T1_ET01 AND NOT #EstadoZona.ParoBlando_CBx AND ((#AVTF_Ent_M1 AND #Avance_13) OR (NOT #AVTF_Ent_M1 AND NOT #AVTF_Ent_M2 AND NOT #AVTF_Ent_M4 AND #pHsMx)) AND #EstadoZona.Marcha_CBx AND NOT #O_Sal_S3 AND NOT #O_Sal_S4 AND NOT #O_Vaciar AND NOT #T1_ET50 AND NOT #T1_ET02 THEN
       #T1_ET10 := TRUE;   // SR flip-flop
   END_IF;
   IF #T1_ET11 THEN #T1_ET10 := FALSE; END_IF;
END_REGION

REGION Network 21: #T1_ET20.
   RUNG wire#powerrail
      Contact( #T1_ET01 )
      I_Contact( #EstadoZona.ParoBlando_CBx )
      wire#w1
      Contact( #Selec_M2_Entrada )
      wire#w2
      Contact( #PosTR_E2 )
      Contact( #EstadoZona.Marcha_CBx )
      I_Contact( #EstadoZona.ParoBlando_CBx )
      I_Contact( #O_Sal_S3 )
      I_Contact( #O_Sal_S4 )
      I_Contact( #O_Vaciar )
      I_Contact( #T1_ET50 )
      I_Contact( #T1_ET02 )
      S_SR(operand := #T1_ET20, r1 := #T1_ET21)
   END_RUNG
   RUNG wire#w1
      Contact( #Selec_M4_Entrada )
   END_RUNG wire#w2
   // the same network as SCL:
   IF #T1_ET01 AND NOT #EstadoZona.ParoBlando_CBx AND (#Selec_M2_Entrada OR #Selec_M4_Entrada) AND #PosTR_E2 AND #EstadoZona.Marcha_CBx AND NOT #EstadoZona.ParoBlando_CBx AND NOT #O_Sal_S3 AND NOT #O_Sal_S4 AND NOT #O_Vaciar AND NOT #T1_ET50 AND NOT #T1_ET02 THEN
       #T1_ET20 := TRUE;   // SR flip-flop
   END_IF;
   IF #T1_ET21 THEN #T1_ET20 := FALSE; END_IF;
END_REGION

REGION Network 22: #CNT_Aus_S4
   RUNG wire#powerrail
      "FC912_CNT_Tiempo_Mem_UHS"(Temporizar := wire#w1, Reset := wire#w2, Valor_Tiempo := #V_CNT_ApHsMx_S4, Base_tiempo_ms := 1, Valor_Actual := #TMP_Aus_S4, Tiempo_OK => #tmp_Aus_S4_Q)
   END_RUNG
   RUNG wire#powerrail
      Contact( #T1_ET60 )
      Contact( "DB1_SalidasExterioresDeMesa".Mesa[#Mesa].Avanzar_E2E4 )
      Contact( #PosTR_E2 )
      I_Contact( #pHsMx )
   END_RUNG wire#w1
   RUNG wire#powerrail
      I_Contact( #T1_ET60 )
   END_RUNG wire#w2
   // the same network as SCL:
   "FC912_CNT_Tiempo_Mem_UHS"(Temporizar := #T1_ET60 AND "DB1_SalidasExterioresDeMesa".Mesa[#Mesa].Avanzar_E2E4 AND #PosTR_E2 AND NOT #pHsMx,
                           Reset := NOT #T1_ET60,
                           Valor_Tiempo := #V_CNT_ApHsMx_S4,
                           Base_tiempo_ms := 1,
                           Valor_Actual := #TMP_Aus_S4,
                           Tiempo_OK => #tmp_Aus_S4_Q);
END_REGION

REGION Network 23: #TMP_Aus_S3
   RUNG wire#powerrail
      "FC912_CNT_Tiempo_Mem_UHS"(Temporizar := wire#w3, Reset := wire#w4, Valor_Tiempo := #V_CNT_ApHsMx_S3, Base_tiempo_ms := 1, Valor_Actual := #TMP_Aus_S3, Tiempo_OK => #tmp_pHs_S3_Q)
   END_RUNG
   RUNG wire#powerrail
      Contact( #T1_ET50 )
      Contact( #Avance_13 )
      wire#w1
      Contact( #NXT_Avance_S3 )
      wire#w2
      Contact( #PosTR_E1 )
      I_Contact( #pHsMx )
   END_RUNG wire#w3
   RUNG wire#w1
      Contact( #PTF_Sal_M3 )
   END_RUNG wire#w2
   RUNG wire#powerrail
      I_Contact( #T1_ET50 )
   END_RUNG wire#w4
   // the same network as SCL:
   "FC912_CNT_Tiempo_Mem_UHS"(Temporizar := #T1_ET50 AND #Avance_13 AND (#NXT_Avance_S3 OR #PTF_Sal_M3) AND #PosTR_E1 AND NOT #pHsMx,
                           Reset := NOT #T1_ET50,
                           Valor_Tiempo := #V_CNT_ApHsMx_S3,
                           Base_tiempo_ms := 1,
                           Valor_Actual := #TMP_Aus_S3,
                           Tiempo_OK => #tmp_pHs_S3_Q);
END_REGION

REGION Network 24: #T1_ET01. ESTADO REPOSO VACIO.
   RUNG wire#powerrail
      Contact( #T1_ET00 )
      I_Contact( #pHsMx )
      Contact( #EstadoZona.Marcha_CBx )
      wire#w1
      S_SR(operand := #T1_ET01, r1 := wire#w4)
   END_RUNG
   RUNG wire#powerrail
      Contact( #T1_ET50 )
      Contact( #tmp_pHs_S3_Q )
      wire#w2
      Contact( #TRANS_OK )
   END_RUNG wire#w1
   RUNG wire#powerrail
      Contact( #T1_ET60 )
      Contact( #tmp_Aus_S4_Q )
   END_RUNG wire#w2
   RUNG wire#powerrail
      Contact( #T1_ET10 )
      wire#w3
      Contact( #T1_ET110 )
   END_RUNG wire#w4
   RUNG wire#powerrail
      Contact( #T1_ET20 )
   END_RUNG wire#w3
   RUNG wire#powerrail
      Contact( #T1_ET03 )
   END_RUNG wire#w4
   // the same network as SCL:
   IF (#T1_ET00 AND NOT #pHsMx AND #EstadoZona.Marcha_CBx) OR (((#T1_ET50 AND #tmp_pHs_S3_Q) OR (#T1_ET60 AND #tmp_Aus_S4_Q)) AND #TRANS_OK) THEN
       #T1_ET01 := TRUE;   // SR flip-flop
   END_IF;
   IF ((#T1_ET10 OR #T1_ET20) AND #T1_ET110) OR #T1_ET03 THEN #T1_ET01 := FALSE; END_IF;
END_REGION

REGION Network 25: #T1_ET00
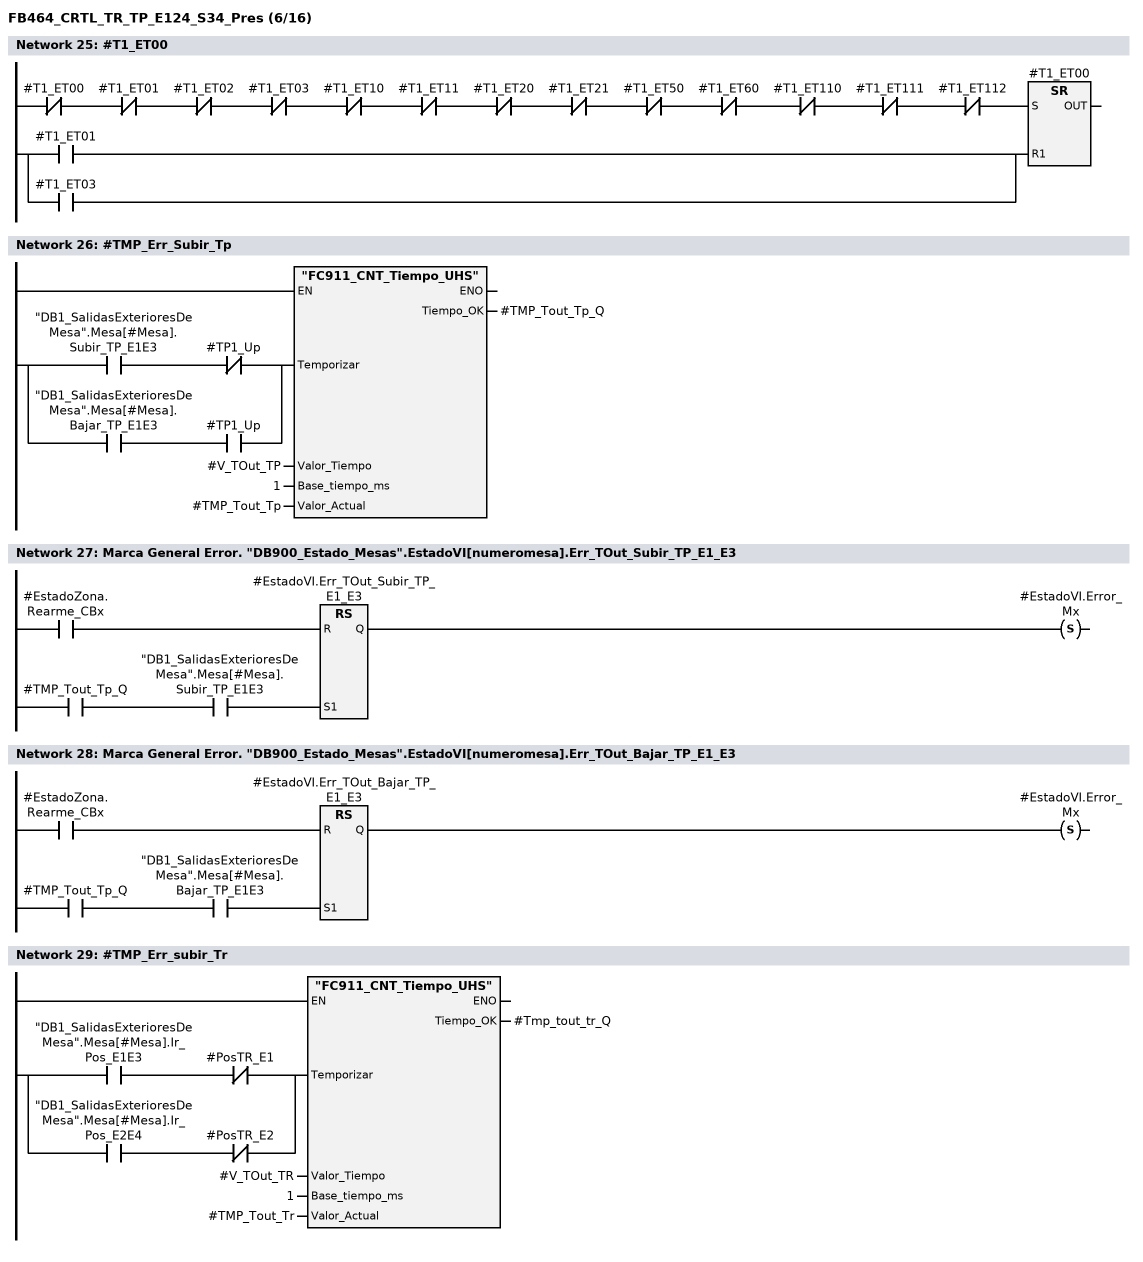
   RUNG wire#powerrail
      I_Contact( #T1_ET00 )
      I_Contact( #T1_ET01 )
      I_Contact( #T1_ET02 )
      I_Contact( #T1_ET03 )
      I_Contact( #T1_ET10 )
      I_Contact( #T1_ET11 )
      I_Contact( #T1_ET20 )
      I_Contact( #T1_ET21 )
      I_Contact( #T1_ET50 )
      I_Contact( #T1_ET60 )
      I_Contact( #T1_ET110 )
      I_Contact( #T1_ET111 )
      I_Contact( #T1_ET112 )
      S_SR(operand := #T1_ET00, r1 := wire#w1)
   END_RUNG
   RUNG wire#powerrail
      Contact( #T1_ET01 )
   END_RUNG wire#w1
   RUNG wire#powerrail
      Contact( #T1_ET03 )
   END_RUNG wire#w1
   // the same network as SCL:
   IF NOT #T1_ET00 AND NOT #T1_ET01 AND NOT #T1_ET02 AND NOT #T1_ET03 AND NOT #T1_ET10 AND NOT #T1_ET11 AND NOT #T1_ET20 AND NOT #T1_ET21 AND NOT #T1_ET50 AND NOT #T1_ET60 AND NOT #T1_ET110 AND NOT #T1_ET111 AND NOT #T1_ET112 THEN
       #T1_ET00 := TRUE;   // SR flip-flop
   END_IF;
   IF #T1_ET01 OR #T1_ET03 THEN #T1_ET00 := FALSE; END_IF;
END_REGION

REGION Network 26: #TMP_Err_Subir_Tp
   RUNG wire#powerrail
      "FC911_CNT_Tiempo_UHS"(Temporizar := wire#w1, Valor_Tiempo := #V_TOut_TP, Base_tiempo_ms := 1, Valor_Actual := #TMP_Tout_Tp, Tiempo_OK => #TMP_Tout_Tp_Q)
   END_RUNG
   RUNG wire#powerrail
      Contact( "DB1_SalidasExterioresDeMesa".Mesa[#Mesa].Subir_TP_E1E3 )
      I_Contact( #TP1_Up )
   END_RUNG wire#w1
   RUNG wire#powerrail
      Contact( "DB1_SalidasExterioresDeMesa".Mesa[#Mesa].Bajar_TP_E1E3 )
      Contact( #TP1_Up )
   END_RUNG wire#w1
   // the same network as SCL:
   "FC911_CNT_Tiempo_UHS"(Temporizar := ("DB1_SalidasExterioresDeMesa".Mesa[#Mesa].Subir_TP_E1E3 AND NOT #TP1_Up) OR ("DB1_SalidasExterioresDeMesa".Mesa[#Mesa].Bajar_TP_E1E3 AND #TP1_Up),
                          Valor_Tiempo := #V_TOut_TP,
                          Base_tiempo_ms := 1,
                          Valor_Actual := #TMP_Tout_Tp,
                          Tiempo_OK => #TMP_Tout_Tp_Q);
END_REGION

REGION Network 27: Marca General Error. "DB900_Estado_Mesas".EstadoVI[numeromesa].Err_TOut_Subir_TP_E1_E3
   RUNG wire#powerrail
      Contact( #EstadoZona.Rearme_CBx )
      S_RS(operand := #EstadoVI.Err_TOut_Subir_TP_E1_E3, s1 := wire#w1)
      S_Coil( #EstadoVI.Error_Mx )
   END_RUNG
   RUNG wire#powerrail
      Contact( #TMP_Tout_Tp_Q )
      Contact( "DB1_SalidasExterioresDeMesa".Mesa[#Mesa].Subir_TP_E1E3 )
   END_RUNG wire#w1
   // the same network as SCL:
   IF #EstadoZona.Rearme_CBx THEN
       #EstadoVI.Err_TOut_Subir_TP_E1_E3 := FALSE;   // RS flip-flop
   END_IF;
   IF #TMP_Tout_Tp_Q AND "DB1_SalidasExterioresDeMesa".Mesa[#Mesa].Subir_TP_E1E3 THEN
       #EstadoVI.Err_TOut_Subir_TP_E1_E3 := TRUE;
   END_IF;
   IF #EstadoVI.Err_TOut_Subir_TP_E1_E3 THEN #EstadoVI.Error_Mx := TRUE; END_IF;
END_REGION

REGION Network 28: Marca General Error. "DB900_Estado_Mesas".EstadoVI[numeromesa].Err_TOut_Bajar_TP_E1_E3
   RUNG wire#powerrail
      Contact( #EstadoZona.Rearme_CBx )
      S_RS(operand := #EstadoVI.Err_TOut_Bajar_TP_E1_E3, s1 := wire#w1)
      S_Coil( #EstadoVI.Error_Mx )
   END_RUNG
   RUNG wire#powerrail
      Contact( #TMP_Tout_Tp_Q )
      Contact( "DB1_SalidasExterioresDeMesa".Mesa[#Mesa].Bajar_TP_E1E3 )
   END_RUNG wire#w1
   // the same network as SCL:
   IF #EstadoZona.Rearme_CBx THEN
       #EstadoVI.Err_TOut_Bajar_TP_E1_E3 := FALSE;   // RS flip-flop
   END_IF;
   IF #TMP_Tout_Tp_Q AND "DB1_SalidasExterioresDeMesa".Mesa[#Mesa].Bajar_TP_E1E3 THEN
       #EstadoVI.Err_TOut_Bajar_TP_E1_E3 := TRUE;
   END_IF;
   IF #EstadoVI.Err_TOut_Bajar_TP_E1_E3 THEN #EstadoVI.Error_Mx := TRUE; END_IF;
END_REGION

REGION Network 29: #TMP_Err_subir_Tr
   RUNG wire#powerrail
      "FC911_CNT_Tiempo_UHS"(Temporizar := wire#w1, Valor_Tiempo := #V_TOut_TR, Base_tiempo_ms := 1, Valor_Actual := #TMP_Tout_Tr, Tiempo_OK => #Tmp_tout_tr_Q)
   END_RUNG
   RUNG wire#powerrail
      Contact( "DB1_SalidasExterioresDeMesa".Mesa[#Mesa].Ir_Pos_E1E3 )
      I_Contact( #PosTR_E1 )
   END_RUNG wire#w1
   RUNG wire#powerrail
      Contact( "DB1_SalidasExterioresDeMesa".Mesa[#Mesa].Ir_Pos_E2E4 )
      I_Contact( #PosTR_E2 )
   END_RUNG wire#w1
   // the same network as SCL:
   "FC911_CNT_Tiempo_UHS"(Temporizar := ("DB1_SalidasExterioresDeMesa".Mesa[#Mesa].Ir_Pos_E1E3 AND NOT #PosTR_E1) OR ("DB1_SalidasExterioresDeMesa".Mesa[#Mesa].Ir_Pos_E2E4 AND NOT #PosTR_E2),
                          Valor_Tiempo := #V_TOut_TR,
                          Base_tiempo_ms := 1,
                          Valor_Actual := #TMP_Tout_Tr,
                          Tiempo_OK => #Tmp_tout_tr_Q);
END_REGION

REGION Network 30: Marca General Error. "DB900_Estado_Mesas".EstadoVI[numeromesa].Err_TOut_Subida
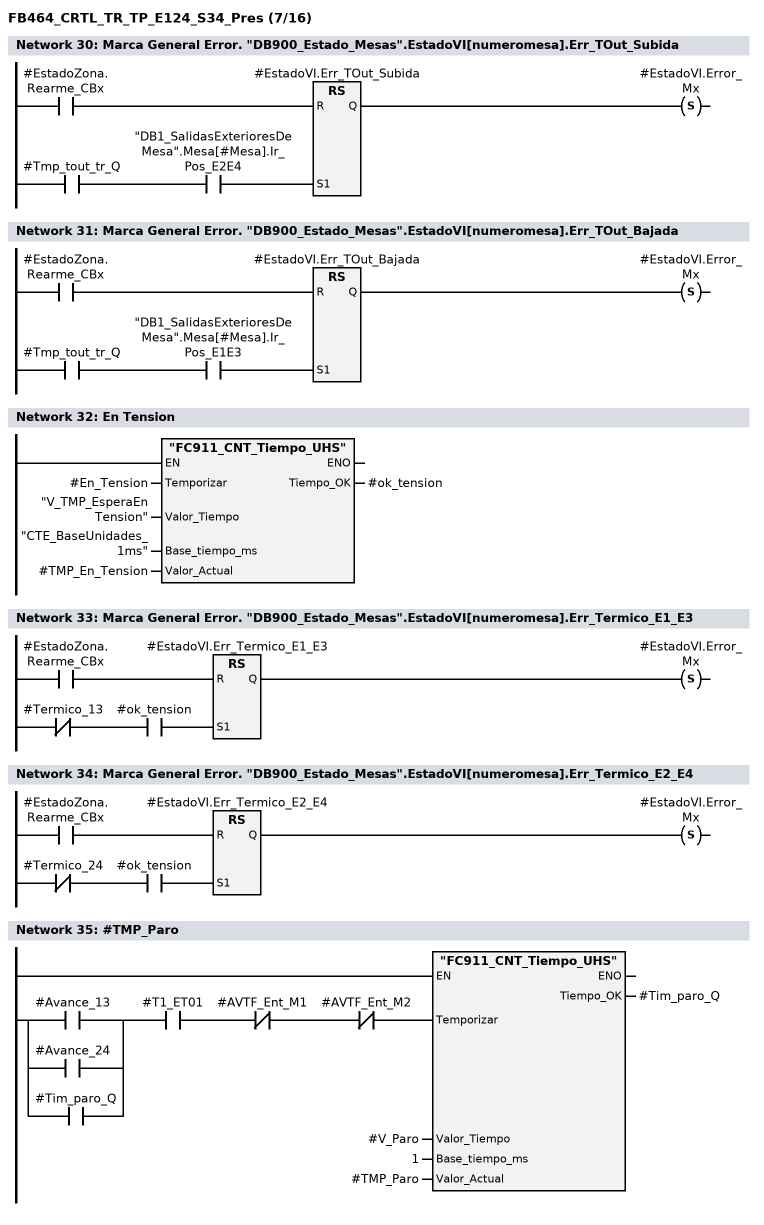
   RUNG wire#powerrail
      Contact( #EstadoZona.Rearme_CBx )
      S_RS(operand := #EstadoVI.Err_TOut_Subida, s1 := wire#w1)
      S_Coil( #EstadoVI.Error_Mx )
   END_RUNG
   RUNG wire#powerrail
      Contact( #Tmp_tout_tr_Q )
      Contact( "DB1_SalidasExterioresDeMesa".Mesa[#Mesa].Ir_Pos_E2E4 )
   END_RUNG wire#w1
   // the same network as SCL:
   IF #EstadoZona.Rearme_CBx THEN
       #EstadoVI.Err_TOut_Subida := FALSE;   // RS flip-flop
   END_IF;
   IF #Tmp_tout_tr_Q AND "DB1_SalidasExterioresDeMesa".Mesa[#Mesa].Ir_Pos_E2E4 THEN
       #EstadoVI.Err_TOut_Subida := TRUE;
   END_IF;
   IF #EstadoVI.Err_TOut_Subida THEN #EstadoVI.Error_Mx := TRUE; END_IF;
END_REGION

REGION Network 31: Marca General Error. "DB900_Estado_Mesas".EstadoVI[numeromesa].Err_TOut_Bajada
   RUNG wire#powerrail
      Contact( #EstadoZona.Rearme_CBx )
      S_RS(operand := #EstadoVI.Err_TOut_Bajada, s1 := wire#w1)
      S_Coil( #EstadoVI.Error_Mx )
   END_RUNG
   RUNG wire#powerrail
      Contact( #Tmp_tout_tr_Q )
      Contact( "DB1_SalidasExterioresDeMesa".Mesa[#Mesa].Ir_Pos_E1E3 )
   END_RUNG wire#w1
   // the same network as SCL:
   IF #EstadoZona.Rearme_CBx THEN
       #EstadoVI.Err_TOut_Bajada := FALSE;   // RS flip-flop
   END_IF;
   IF #Tmp_tout_tr_Q AND "DB1_SalidasExterioresDeMesa".Mesa[#Mesa].Ir_Pos_E1E3 THEN
       #EstadoVI.Err_TOut_Bajada := TRUE;
   END_IF;
   IF #EstadoVI.Err_TOut_Bajada THEN #EstadoVI.Error_Mx := TRUE; END_IF;
END_REGION

REGION Network 32: En Tension
   RUNG wire#powerrail
      "FC911_CNT_Tiempo_UHS"(Temporizar := #En_Tension, Valor_Tiempo := "V_TMP_EsperaEnTension", Base_tiempo_ms := "CTE_BaseUnidades_1ms", Valor_Actual := #TMP_En_Tension, Tiempo_OK => #ok_tension)
   END_RUNG
   // the same network as SCL:
   "FC911_CNT_Tiempo_UHS"(Temporizar := #En_Tension,
                          Valor_Tiempo := "V_TMP_EsperaEnTension",
                          Base_tiempo_ms := "CTE_BaseUnidades_1ms",
                          Valor_Actual := #TMP_En_Tension,
                          Tiempo_OK => #ok_tension);
END_REGION

REGION Network 33: Marca General Error. "DB900_Estado_Mesas".EstadoVI[numeromesa].Err_Termico_E1_E3
   RUNG wire#powerrail
      Contact( #EstadoZona.Rearme_CBx )
      S_RS(operand := #EstadoVI.Err_Termico_E1_E3, s1 := wire#w1)
      S_Coil( #EstadoVI.Error_Mx )
   END_RUNG
   RUNG wire#powerrail
      I_Contact( #Termico_13 )
      Contact( #ok_tension )
   END_RUNG wire#w1
   // the same network as SCL:
   IF #EstadoZona.Rearme_CBx THEN
       #EstadoVI.Err_Termico_E1_E3 := FALSE;   // RS flip-flop
   END_IF;
   IF NOT #Termico_13 AND #ok_tension THEN #EstadoVI.Err_Termico_E1_E3 := TRUE; END_IF;
   IF #EstadoVI.Err_Termico_E1_E3 THEN #EstadoVI.Error_Mx := TRUE; END_IF;
END_REGION

REGION Network 34: Marca General Error. "DB900_Estado_Mesas".EstadoVI[numeromesa].Err_Termico_E2_E4
   RUNG wire#powerrail
      Contact( #EstadoZona.Rearme_CBx )
      S_RS(operand := #EstadoVI.Err_Termico_E2_E4, s1 := wire#w1)
      S_Coil( #EstadoVI.Error_Mx )
   END_RUNG
   RUNG wire#powerrail
      I_Contact( #Termico_24 )
      Contact( #ok_tension )
   END_RUNG wire#w1
   // the same network as SCL:
   IF #EstadoZona.Rearme_CBx THEN
       #EstadoVI.Err_Termico_E2_E4 := FALSE;   // RS flip-flop
   END_IF;
   IF NOT #Termico_24 AND #ok_tension THEN #EstadoVI.Err_Termico_E2_E4 := TRUE; END_IF;
   IF #EstadoVI.Err_Termico_E2_E4 THEN #EstadoVI.Error_Mx := TRUE; END_IF;
END_REGION

REGION Network 35: #TMP_Paro
   RUNG wire#powerrail
      "FC911_CNT_Tiempo_UHS"(Temporizar := wire#w2, Valor_Tiempo := #V_Paro, Base_tiempo_ms := 1, Valor_Actual := #TMP_Paro, Tiempo_OK => #Tim_paro_Q)
   END_RUNG
   RUNG wire#powerrail
      Contact( #Avance_13 )
      wire#w1
      Contact( #T1_ET01 )
      I_Contact( #AVTF_Ent_M1 )
      I_Contact( #AVTF_Ent_M2 )
   END_RUNG wire#w2
   RUNG wire#powerrail
      Contact( #Avance_24 )
   END_RUNG wire#w1
   RUNG wire#powerrail
      Contact( #Tim_paro_Q )
   END_RUNG wire#w1
   // the same network as SCL:
   "FC911_CNT_Tiempo_UHS"(Temporizar := (#Avance_13 OR #Avance_24 OR #Tim_paro_Q) AND #T1_ET01 AND NOT #AVTF_Ent_M1 AND NOT #AVTF_Ent_M2,
                          Valor_Tiempo := #V_Paro,
                          Base_tiempo_ms := 1,
                          Valor_Actual := #TMP_Paro,
                          Tiempo_OK => #Tim_paro_Q);
END_REGION

REGION Network 36: tout avance
   // Nieves 16/12/17. incluyo porque no existe el error
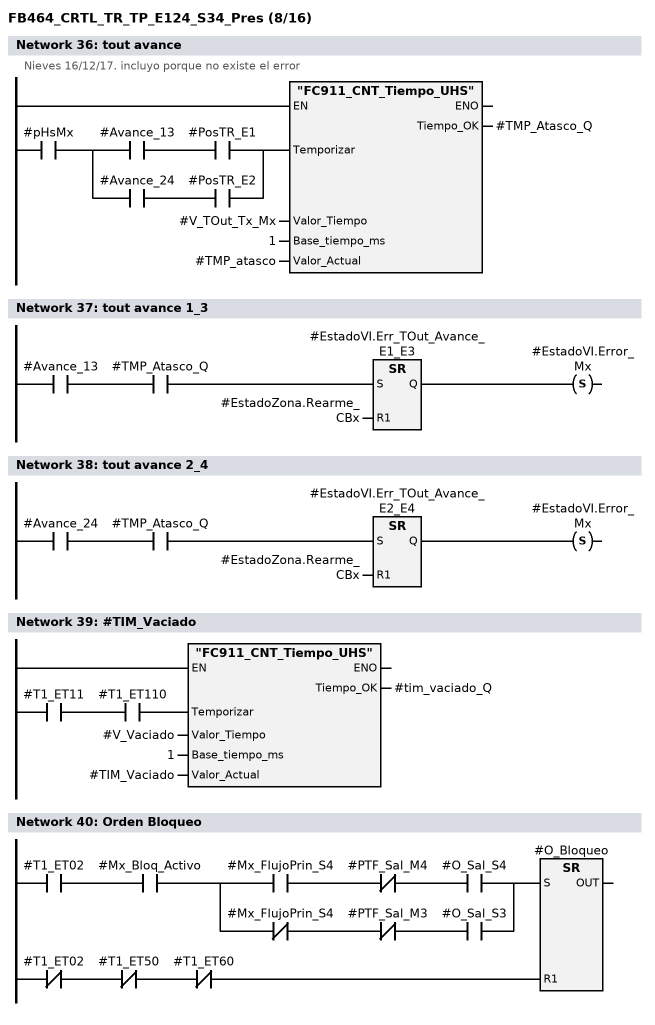
   RUNG wire#powerrail
      "FC911_CNT_Tiempo_UHS"(Temporizar := wire#w2, Valor_Tiempo := #V_TOut_Tx_Mx, Base_tiempo_ms := 1, Valor_Actual := #TMP_atasco, Tiempo_OK => #TMP_Atasco_Q)
   END_RUNG
   RUNG wire#powerrail
      Contact( #pHsMx )
      wire#w1
      Contact( #Avance_13 )
      Contact( #PosTR_E1 )
   END_RUNG wire#w2
   RUNG wire#w1
      Contact( #Avance_24 )
      Contact( #PosTR_E2 )
   END_RUNG wire#w2
   // the same network as SCL:
   "FC911_CNT_Tiempo_UHS"(Temporizar := #pHsMx AND ((#Avance_13 AND #PosTR_E1) OR (#Avance_24 AND #PosTR_E2)),
                          Valor_Tiempo := #V_TOut_Tx_Mx,
                          Base_tiempo_ms := 1,
                          Valor_Actual := #TMP_atasco,
                          Tiempo_OK => #TMP_Atasco_Q);
END_REGION

REGION Network 37: tout avance 1_3
   RUNG wire#powerrail
      Contact( #Avance_13 )
      Contact( #TMP_Atasco_Q )
      S_SR(operand := #EstadoVI.Err_TOut_Avance_E1_E3, r1 := #EstadoZona.Rearme_CBx)
      S_Coil( #EstadoVI.Error_Mx )
   END_RUNG
   // the same network as SCL:
   IF #Avance_13 AND #TMP_Atasco_Q THEN
       #EstadoVI.Err_TOut_Avance_E1_E3 := TRUE;   // SR flip-flop
   END_IF;
   IF #EstadoZona.Rearme_CBx THEN #EstadoVI.Err_TOut_Avance_E1_E3 := FALSE; END_IF;
   IF #EstadoVI.Err_TOut_Avance_E1_E3 THEN #EstadoVI.Error_Mx := TRUE; END_IF;
END_REGION

REGION Network 38: tout avance 2_4
   RUNG wire#powerrail
      Contact( #Avance_24 )
      Contact( #TMP_Atasco_Q )
      S_SR(operand := #EstadoVI.Err_TOut_Avance_E2_E4, r1 := #EstadoZona.Rearme_CBx)
      S_Coil( #EstadoVI.Error_Mx )
   END_RUNG
   // the same network as SCL:
   IF #Avance_24 AND #TMP_Atasco_Q THEN
       #EstadoVI.Err_TOut_Avance_E2_E4 := TRUE;   // SR flip-flop
   END_IF;
   IF #EstadoZona.Rearme_CBx THEN #EstadoVI.Err_TOut_Avance_E2_E4 := FALSE; END_IF;
   IF #EstadoVI.Err_TOut_Avance_E2_E4 THEN #EstadoVI.Error_Mx := TRUE; END_IF;
END_REGION

REGION Network 39: #TIM_Vaciado
   RUNG wire#powerrail
      "FC911_CNT_Tiempo_UHS"(Temporizar := wire#w1, Valor_Tiempo := #V_Vaciado, Base_tiempo_ms := 1, Valor_Actual := #TIM_Vaciado, Tiempo_OK => #tim_vaciado_Q)
   END_RUNG
   RUNG wire#powerrail
      Contact( #T1_ET11 )
      Contact( #T1_ET110 )
   END_RUNG wire#w1
   // the same network as SCL:
   "FC911_CNT_Tiempo_UHS"(Temporizar := #T1_ET11 AND #T1_ET110,
                          Valor_Tiempo := #V_Vaciado,
                          Base_tiempo_ms := 1,
                          Valor_Actual := #TIM_Vaciado,
                          Tiempo_OK => #tim_vaciado_Q);
END_REGION

REGION Network 40: Orden Bloqueo
   RUNG wire#powerrail
      Contact( #T1_ET02 )
      Contact( #Mx_Bloq_Activo )
      wire#w1
      Contact( #Mx_FlujoPrin_S4 )
      I_Contact( #PTF_Sal_M4 )
      Contact( #O_Sal_S4 )
      wire#w2
      S_SR(operand := #O_Bloqueo, r1 := wire#w3)
   END_RUNG
   RUNG wire#w1
      I_Contact( #Mx_FlujoPrin_S4 )
      I_Contact( #PTF_Sal_M3 )
      Contact( #O_Sal_S3 )
   END_RUNG wire#w2
   RUNG wire#powerrail
      I_Contact( #T1_ET02 )
      I_Contact( #T1_ET50 )
      I_Contact( #T1_ET60 )
   END_RUNG wire#w3
   // the same network as SCL:
   IF #T1_ET02 AND #Mx_Bloq_Activo AND ((#Mx_FlujoPrin_S4 AND NOT #PTF_Sal_M4 AND #O_Sal_S4) OR (NOT #Mx_FlujoPrin_S4 AND NOT #PTF_Sal_M3 AND #O_Sal_S3)) THEN
       #O_Bloqueo := TRUE;   // SR flip-flop
   END_IF;
   IF NOT #T1_ET02 AND NOT #T1_ET50 AND NOT #T1_ET60 THEN #O_Bloqueo := FALSE; END_IF;
END_REGION

REGION Network 41: Subir Tope
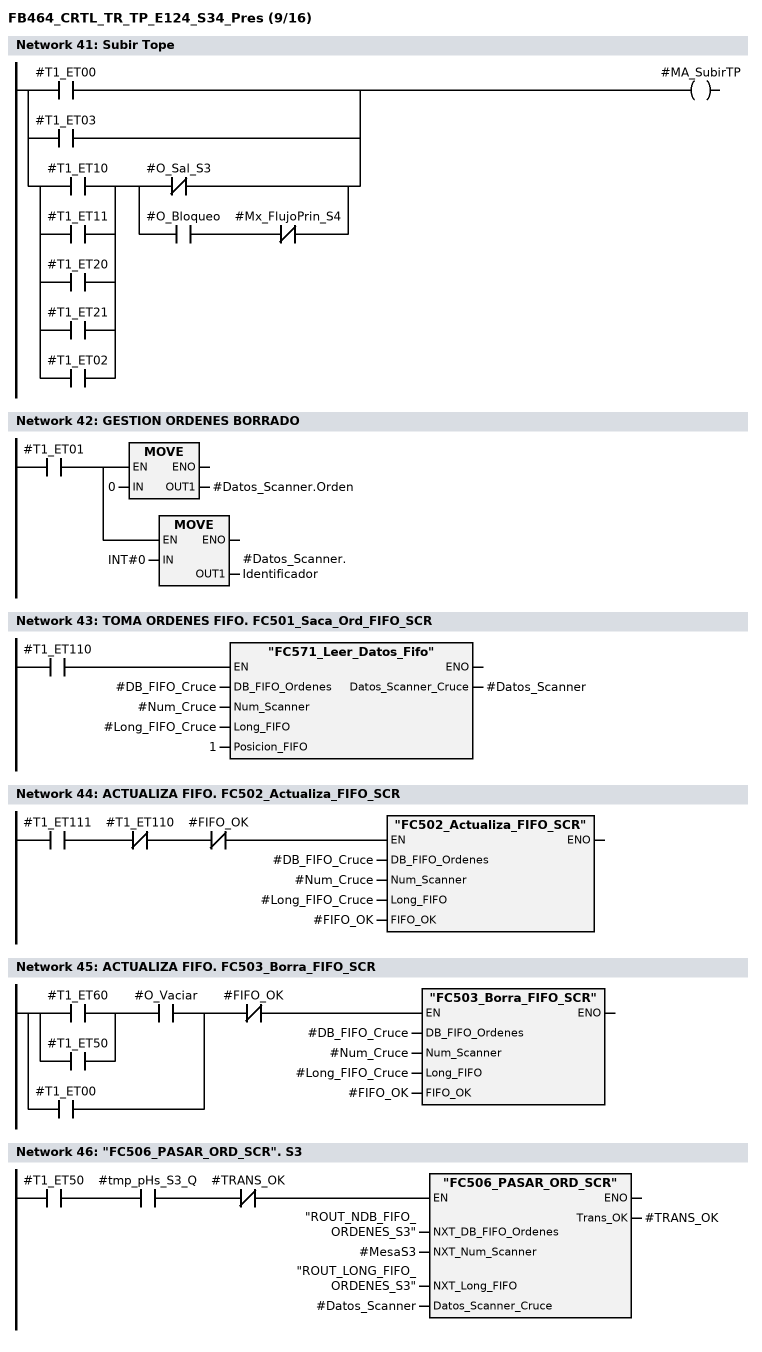
   RUNG wire#powerrail
      Contact( #T1_ET00 )
      wire#w1
      Coil( #MA_SubirTP )
   END_RUNG
   RUNG wire#powerrail
      Contact( #T1_ET03 )
   END_RUNG wire#w1
   RUNG wire#powerrail
      Contact( #T1_ET10 )
      wire#w2
      I_Contact( #O_Sal_S3 )
   END_RUNG wire#w1
   RUNG wire#powerrail
      Contact( #T1_ET11 )
   END_RUNG wire#w2
   RUNG wire#powerrail
      Contact( #T1_ET20 )
   END_RUNG wire#w2
   RUNG wire#powerrail
      Contact( #T1_ET21 )
   END_RUNG wire#w2
   RUNG wire#powerrail
      Contact( #T1_ET02 )
   END_RUNG wire#w2
   RUNG wire#w2
      Contact( #O_Bloqueo )
      I_Contact( #Mx_FlujoPrin_S4 )
   END_RUNG wire#w1
   // the same network as SCL:
   #MA_SubirTP := #T1_ET00 OR #T1_ET03 OR ((#T1_ET10 OR #T1_ET11 OR #T1_ET20 OR #T1_ET21 OR #T1_ET02) AND (NOT #O_Sal_S3 OR (#O_Bloqueo AND NOT #Mx_FlujoPrin_S4)));
END_REGION

REGION Network 42: GESTION ORDENES BORRADO
   RUNG wire#powerrail
      Contact( #T1_ET01 )
      wire#w1
      { S7_GenerateENO := "TRUE" } Move(in := 0, out1 => #Datos_Scanner.Orden)
   END_RUNG
   RUNG wire#w1
      { S7_GenerateENO := "TRUE" } Move(in := INT#0, out1 => #Datos_Scanner.Identificador)
   END_RUNG
   // the same network as SCL:
   IF #T1_ET01 THEN
       #Datos_Scanner.Orden := 0;
       #Datos_Scanner.Identificador := INT#0;
   END_IF;
END_REGION

REGION Network 43: TOMA ORDENES FIFO. FC501_Saca_Ord_FIFO_SCR
   RUNG wire#powerrail
      Contact( #T1_ET110 )
      "FC571_Leer_Datos_Fifo"(DB_FIFO_Ordenes := #DB_FIFO_Cruce, Num_Scanner := #Num_Cruce, Long_FIFO := #Long_FIFO_Cruce, Posicion_FIFO := 1, Datos_Scanner_Cruce => #Datos_Scanner)
   END_RUNG
   // the same network as SCL:
   IF #T1_ET110 THEN
       "FC571_Leer_Datos_Fifo"(DB_FIFO_Ordenes := #DB_FIFO_Cruce,
                               Num_Scanner := #Num_Cruce,
                               Long_FIFO := #Long_FIFO_Cruce,
                               Posicion_FIFO := 1,
                               Datos_Scanner_Cruce => #Datos_Scanner);
   END_IF;
END_REGION

REGION Network 44: ACTUALIZA FIFO. FC502_Actualiza_FIFO_SCR
   RUNG wire#powerrail
      Contact( #T1_ET111 )
      I_Contact( #T1_ET110 )
      I_Contact( #FIFO_OK )
      "FC502_Actualiza_FIFO_SCR"(DB_FIFO_Ordenes := #DB_FIFO_Cruce, Num_Scanner := #Num_Cruce, Long_FIFO := #Long_FIFO_Cruce, FIFO_OK := #FIFO_OK)
   END_RUNG
   // the same network as SCL:
   IF #T1_ET111 AND NOT #T1_ET110 AND NOT #FIFO_OK THEN
       "FC502_Actualiza_FIFO_SCR"(DB_FIFO_Ordenes := #DB_FIFO_Cruce,
                               Num_Scanner := #Num_Cruce,
                               Long_FIFO := #Long_FIFO_Cruce,
                               FIFO_OK := #FIFO_OK);
   END_IF;
END_REGION

REGION Network 45: ACTUALIZA FIFO. FC503_Borra_FIFO_SCR
   RUNG wire#powerrail
      Contact( #T1_ET60 )
      wire#w1
      Contact( #O_Vaciar )
      wire#w2
      I_Contact( #FIFO_OK )
      "FC503_Borra_FIFO_SCR"(DB_FIFO_Ordenes := #DB_FIFO_Cruce, Num_Scanner := #Num_Cruce, Long_FIFO := #Long_FIFO_Cruce, FIFO_OK := #FIFO_OK)
   END_RUNG
   RUNG wire#powerrail
      Contact( #T1_ET50 )
   END_RUNG wire#w1
   RUNG wire#powerrail
      Contact( #T1_ET00 )
   END_RUNG wire#w2
   // the same network as SCL:
   IF (((#T1_ET60 OR #T1_ET50) AND #O_Vaciar) OR #T1_ET00) AND NOT #FIFO_OK THEN
       "FC503_Borra_FIFO_SCR"(DB_FIFO_Ordenes := #DB_FIFO_Cruce,
                              Num_Scanner := #Num_Cruce,
                              Long_FIFO := #Long_FIFO_Cruce,
                              FIFO_OK := #FIFO_OK);
   END_IF;
END_REGION

REGION Network 46: "FC506_PASAR_ORD_SCR". S3
   RUNG wire#powerrail
      Contact( #T1_ET50 )
      Contact( #tmp_pHs_S3_Q )
      I_Contact( #TRANS_OK )
      "FC506_PASAR_ORD_SCR"(NXT_DB_FIFO_Ordenes := "ROUT_NDB_FIFO_ORDENES_S3", NXT_Num_Scanner := #MesaS3, NXT_Long_FIFO := "ROUT_LONG_FIFO_ORDENES_S3", Datos_Scanner_Cruce := #Datos_Scanner, Trans_OK => #TRANS_OK)
   END_RUNG
   // the same network as SCL:
   IF #T1_ET50 AND #tmp_pHs_S3_Q AND NOT #TRANS_OK THEN
       "FC506_PASAR_ORD_SCR"(NXT_DB_FIFO_Ordenes := "ROUT_NDB_FIFO_ORDENES_S3",
                             NXT_Num_Scanner := #MesaS3,
                             NXT_Long_FIFO := "ROUT_LONG_FIFO_ORDENES_S3",
                             Datos_Scanner_Cruce := #Datos_Scanner,
                             Trans_OK => #TRANS_OK);
   END_IF;
END_REGION

REGION Network 47: "FC506_PASAR_ORD_SCR". S2
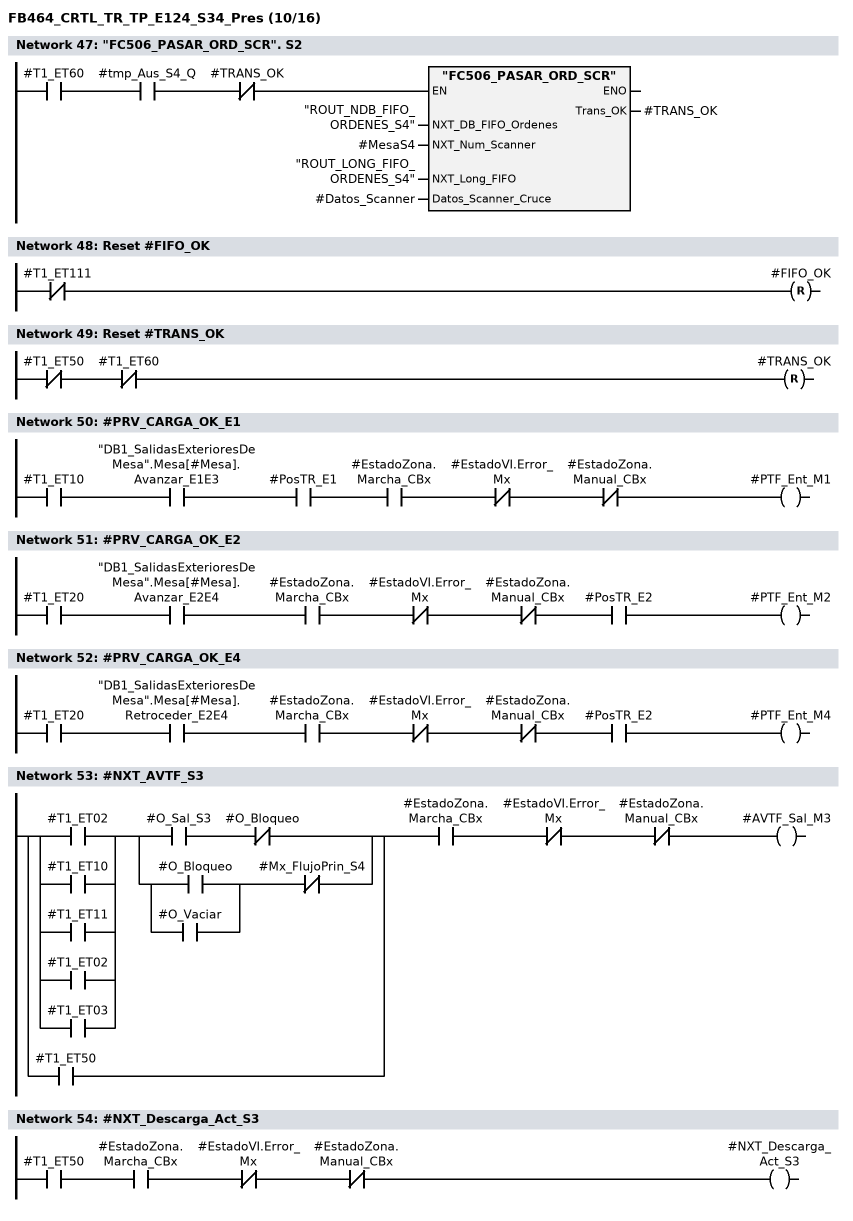
   RUNG wire#powerrail
      Contact( #T1_ET60 )
      Contact( #tmp_Aus_S4_Q )
      I_Contact( #TRANS_OK )
      "FC506_PASAR_ORD_SCR"(NXT_DB_FIFO_Ordenes := "ROUT_NDB_FIFO_ORDENES_S4", NXT_Num_Scanner := #MesaS4, NXT_Long_FIFO := "ROUT_LONG_FIFO_ORDENES_S4", Datos_Scanner_Cruce := #Datos_Scanner, Trans_OK => #TRANS_OK)
   END_RUNG
   // the same network as SCL:
   IF #T1_ET60 AND #tmp_Aus_S4_Q AND NOT #TRANS_OK THEN
       "FC506_PASAR_ORD_SCR"(NXT_DB_FIFO_Ordenes := "ROUT_NDB_FIFO_ORDENES_S4",
                             NXT_Num_Scanner := #MesaS4,
                             NXT_Long_FIFO := "ROUT_LONG_FIFO_ORDENES_S4",
                             Datos_Scanner_Cruce := #Datos_Scanner,
                             Trans_OK => #TRANS_OK);
   END_IF;
END_REGION

REGION Network 48: Reset #FIFO_OK
   RUNG wire#powerrail
      I_Contact( #T1_ET111 )
      R_Coil( #FIFO_OK )
   END_RUNG
   // the same network as SCL:
   IF NOT #T1_ET111 THEN #FIFO_OK := FALSE; END_IF;
END_REGION

REGION Network 49: Reset #TRANS_OK
   RUNG wire#powerrail
      I_Contact( #T1_ET50 )
      I_Contact( #T1_ET60 )
      R_Coil( #TRANS_OK )
   END_RUNG
   // the same network as SCL:
   IF NOT #T1_ET50 AND NOT #T1_ET60 THEN #TRANS_OK := FALSE; END_IF;
END_REGION

REGION Network 50: #PRV_CARGA_OK_E1
   RUNG wire#powerrail
      Contact( #T1_ET10 )
      Contact( "DB1_SalidasExterioresDeMesa".Mesa[#Mesa].Avanzar_E1E3 )
      Contact( #PosTR_E1 )
      Contact( #EstadoZona.Marcha_CBx )
      I_Contact( #EstadoVI.Error_Mx )
      I_Contact( #EstadoZona.Manual_CBx )
      Coil( #PTF_Ent_M1 )
   END_RUNG
   // the same network as SCL:
   #PTF_Ent_M1 := #T1_ET10 AND "DB1_SalidasExterioresDeMesa".Mesa[#Mesa].Avanzar_E1E3 AND #PosTR_E1 AND #EstadoZona.Marcha_CBx AND NOT #EstadoVI.Error_Mx AND NOT #EstadoZona.Manual_CBx;
END_REGION

REGION Network 51: #PRV_CARGA_OK_E2
   RUNG wire#powerrail
      Contact( #T1_ET20 )
      Contact( "DB1_SalidasExterioresDeMesa".Mesa[#Mesa].Avanzar_E2E4 )
      Contact( #EstadoZona.Marcha_CBx )
      I_Contact( #EstadoVI.Error_Mx )
      I_Contact( #EstadoZona.Manual_CBx )
      Contact( #PosTR_E2 )
      Coil( #PTF_Ent_M2 )
   END_RUNG
   // the same network as SCL:
   #PTF_Ent_M2 := #T1_ET20 AND "DB1_SalidasExterioresDeMesa".Mesa[#Mesa].Avanzar_E2E4 AND #EstadoZona.Marcha_CBx AND NOT #EstadoVI.Error_Mx AND NOT #EstadoZona.Manual_CBx AND #PosTR_E2;
END_REGION

REGION Network 52: #PRV_CARGA_OK_E4
   RUNG wire#powerrail
      Contact( #T1_ET20 )
      Contact( "DB1_SalidasExterioresDeMesa".Mesa[#Mesa].Retroceder_E2E4 )
      Contact( #EstadoZona.Marcha_CBx )
      I_Contact( #EstadoVI.Error_Mx )
      I_Contact( #EstadoZona.Manual_CBx )
      Contact( #PosTR_E2 )
      Coil( #PTF_Ent_M4 )
   END_RUNG
   // the same network as SCL:
   #PTF_Ent_M4 := #T1_ET20 AND "DB1_SalidasExterioresDeMesa".Mesa[#Mesa].Retroceder_E2E4 AND #EstadoZona.Marcha_CBx AND NOT #EstadoVI.Error_Mx AND NOT #EstadoZona.Manual_CBx AND #PosTR_E2;
END_REGION

REGION Network 53: #NXT_AVTF_S3
   RUNG wire#powerrail
      Contact( #T1_ET02 )
      wire#w1
      Contact( #O_Sal_S3 )
      I_Contact( #O_Bloqueo )
      wire#w2
      Contact( #EstadoZona.Marcha_CBx )
      I_Contact( #EstadoVI.Error_Mx )
      I_Contact( #EstadoZona.Manual_CBx )
      Coil( #AVTF_Sal_M3 )
   END_RUNG
   RUNG wire#powerrail
      Contact( #T1_ET10 )
   END_RUNG wire#w1
   RUNG wire#powerrail
      Contact( #T1_ET11 )
   END_RUNG wire#w1
   RUNG wire#powerrail
      Contact( #T1_ET02 )
   END_RUNG wire#w1
   RUNG wire#powerrail
      Contact( #T1_ET03 )
   END_RUNG wire#w1
   RUNG wire#w1
      Contact( #O_Bloqueo )
      wire#w3
      I_Contact( #Mx_FlujoPrin_S4 )
   END_RUNG wire#w2
   RUNG wire#w1
      Contact( #O_Vaciar )
   END_RUNG wire#w3
   RUNG wire#powerrail
      Contact( #T1_ET50 )
   END_RUNG wire#w2
   // the same network as SCL:
   #AVTF_Sal_M3 := (((#T1_ET02 OR #T1_ET10 OR #T1_ET11 OR #T1_ET02 OR #T1_ET03) AND ((#O_Sal_S3 AND NOT #O_Bloqueo) OR ((#O_Bloqueo OR #O_Vaciar) AND NOT #Mx_FlujoPrin_S4))) OR #T1_ET50) AND #EstadoZona.Marcha_CBx AND NOT #EstadoVI.Error_Mx AND NOT #EstadoZona.Manual_CBx;
END_REGION

REGION Network 54: #NXT_Descarga_Act_S3
   RUNG wire#powerrail
      Contact( #T1_ET50 )
      Contact( #EstadoZona.Marcha_CBx )
      I_Contact( #EstadoVI.Error_Mx )
      I_Contact( #EstadoZona.Manual_CBx )
      Coil( #NXT_Descarga_Act_S3 )
   END_RUNG
   // the same network as SCL:
   #NXT_Descarga_Act_S3 := #T1_ET50 AND #EstadoZona.Marcha_CBx AND NOT #EstadoVI.Error_Mx AND NOT #EstadoZona.Manual_CBx;
END_REGION

REGION Network 55: #NXT_AVTF_S2
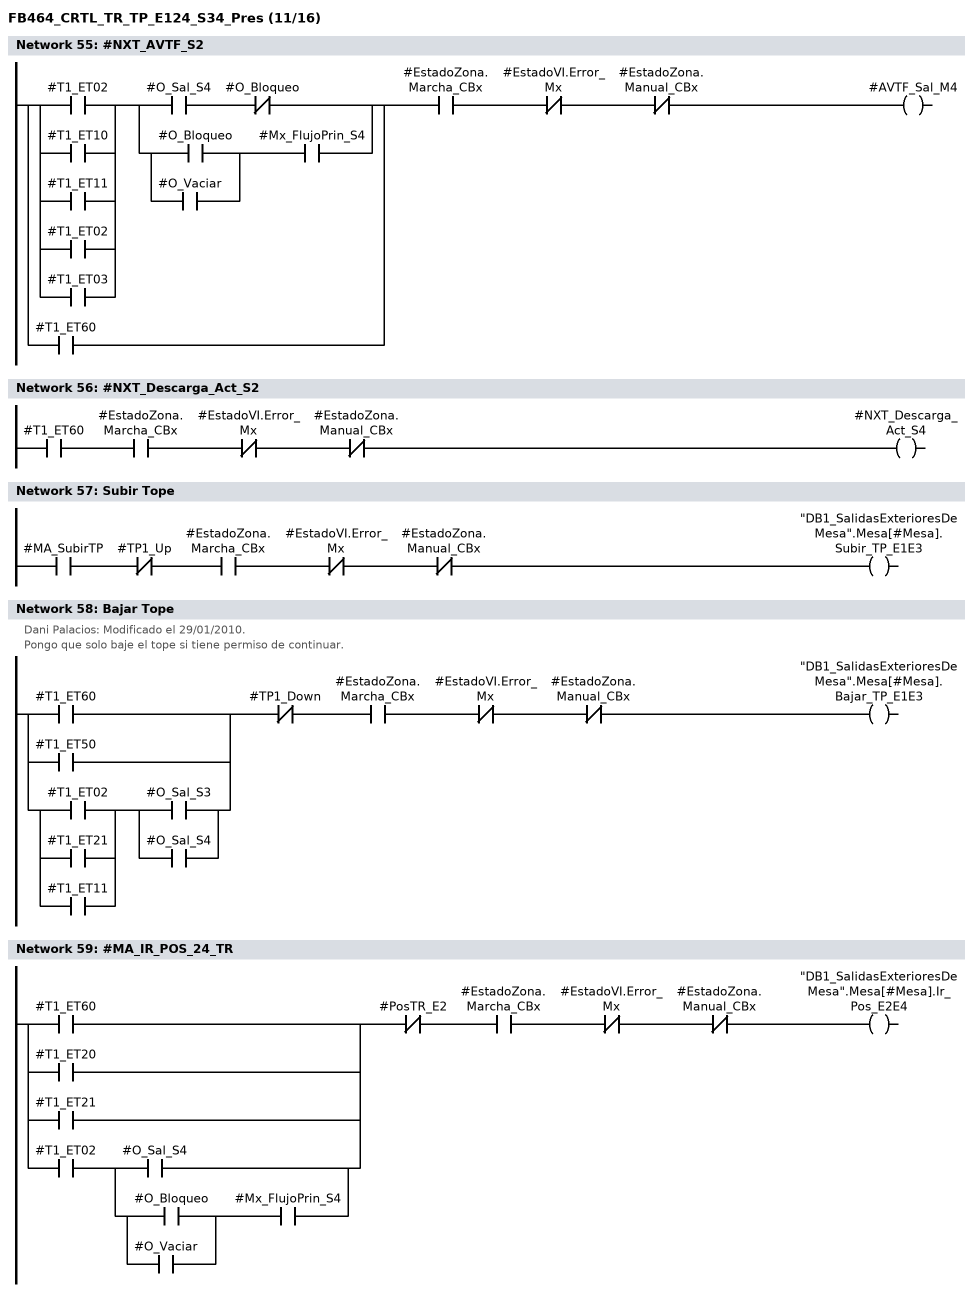
   RUNG wire#powerrail
      Contact( #T1_ET02 )
      wire#w1
      Contact( #O_Sal_S4 )
      I_Contact( #O_Bloqueo )
      wire#w2
      Contact( #EstadoZona.Marcha_CBx )
      I_Contact( #EstadoVI.Error_Mx )
      I_Contact( #EstadoZona.Manual_CBx )
      Coil( #AVTF_Sal_M4 )
   END_RUNG
   RUNG wire#powerrail
      Contact( #T1_ET10 )
   END_RUNG wire#w1
   RUNG wire#powerrail
      Contact( #T1_ET11 )
   END_RUNG wire#w1
   RUNG wire#powerrail
      Contact( #T1_ET02 )
   END_RUNG wire#w1
   RUNG wire#powerrail
      Contact( #T1_ET03 )
   END_RUNG wire#w1
   RUNG wire#w1
      Contact( #O_Bloqueo )
      wire#w3
      Contact( #Mx_FlujoPrin_S4 )
   END_RUNG wire#w2
   RUNG wire#w1
      Contact( #O_Vaciar )
   END_RUNG wire#w3
   RUNG wire#powerrail
      Contact( #T1_ET60 )
   END_RUNG wire#w2
   // the same network as SCL:
   #AVTF_Sal_M4 := (((#T1_ET02 OR #T1_ET10 OR #T1_ET11 OR #T1_ET02 OR #T1_ET03) AND ((#O_Sal_S4 AND NOT #O_Bloqueo) OR ((#O_Bloqueo OR #O_Vaciar) AND #Mx_FlujoPrin_S4))) OR #T1_ET60) AND #EstadoZona.Marcha_CBx AND NOT #EstadoVI.Error_Mx AND NOT #EstadoZona.Manual_CBx;
END_REGION

REGION Network 56: #NXT_Descarga_Act_S2
   RUNG wire#powerrail
      Contact( #T1_ET60 )
      Contact( #EstadoZona.Marcha_CBx )
      I_Contact( #EstadoVI.Error_Mx )
      I_Contact( #EstadoZona.Manual_CBx )
      Coil( #NXT_Descarga_Act_S4 )
   END_RUNG
   // the same network as SCL:
   #NXT_Descarga_Act_S4 := #T1_ET60 AND #EstadoZona.Marcha_CBx AND NOT #EstadoVI.Error_Mx AND NOT #EstadoZona.Manual_CBx;
END_REGION

REGION Network 57: Subir Tope
   RUNG wire#powerrail
      Contact( #MA_SubirTP )
      I_Contact( #TP1_Up )
      Contact( #EstadoZona.Marcha_CBx )
      I_Contact( #EstadoVI.Error_Mx )
      I_Contact( #EstadoZona.Manual_CBx )
      Coil( "DB1_SalidasExterioresDeMesa".Mesa[#Mesa].Subir_TP_E1E3 )
   END_RUNG
   // the same network as SCL:
   "DB1_SalidasExterioresDeMesa".Mesa[#Mesa].Subir_TP_E1E3 := #MA_SubirTP AND NOT #TP1_Up AND #EstadoZona.Marcha_CBx AND NOT #EstadoVI.Error_Mx AND NOT #EstadoZona.Manual_CBx;
END_REGION

REGION Network 58: Bajar Tope
   // Dani Palacios: Modificado el 29/01/2010.
   // Pongo que solo baje el tope si tiene permiso de continuar.
   RUNG wire#powerrail
      Contact( #T1_ET60 )
      wire#w1
      I_Contact( #TP1_Down )
      Contact( #EstadoZona.Marcha_CBx )
      I_Contact( #EstadoVI.Error_Mx )
      I_Contact( #EstadoZona.Manual_CBx )
      Coil( "DB1_SalidasExterioresDeMesa".Mesa[#Mesa].Bajar_TP_E1E3 )
   END_RUNG
   RUNG wire#powerrail
      Contact( #T1_ET50 )
   END_RUNG wire#w1
   RUNG wire#powerrail
      Contact( #T1_ET02 )
      wire#w2
      Contact( #O_Sal_S3 )
   END_RUNG wire#w1
   RUNG wire#powerrail
      Contact( #T1_ET21 )
   END_RUNG wire#w2
   RUNG wire#powerrail
      Contact( #T1_ET11 )
   END_RUNG wire#w2
   RUNG wire#w2
      Contact( #O_Sal_S4 )
   END_RUNG wire#w1
   // the same network as SCL:
   "DB1_SalidasExterioresDeMesa".Mesa[#Mesa].Bajar_TP_E1E3 := (#T1_ET60 OR #T1_ET50 OR ((#T1_ET02 OR #T1_ET21 OR #T1_ET11) AND (#O_Sal_S3 OR #O_Sal_S4))) AND NOT #TP1_Down AND #EstadoZona.Marcha_CBx AND NOT #EstadoVI.Error_Mx AND NOT #EstadoZona.Manual_CBx;
END_REGION

REGION Network 59: #MA_IR_POS_24_TR
   RUNG wire#powerrail
      Contact( #T1_ET60 )
      wire#w1
      I_Contact( #PosTR_E2 )
      Contact( #EstadoZona.Marcha_CBx )
      I_Contact( #EstadoVI.Error_Mx )
      I_Contact( #EstadoZona.Manual_CBx )
      Coil( "DB1_SalidasExterioresDeMesa".Mesa[#Mesa].Ir_Pos_E2E4 )
   END_RUNG
   RUNG wire#powerrail
      Contact( #T1_ET20 )
   END_RUNG wire#w1
   RUNG wire#powerrail
      Contact( #T1_ET21 )
   END_RUNG wire#w1
   RUNG wire#powerrail
      Contact( #T1_ET02 )
      wire#w2
      Contact( #O_Sal_S4 )
   END_RUNG wire#w1
   RUNG wire#w2
      Contact( #O_Bloqueo )
      wire#w3
      Contact( #Mx_FlujoPrin_S4 )
   END_RUNG wire#w1
   RUNG wire#w2
      Contact( #O_Vaciar )
   END_RUNG wire#w3
   // the same network as SCL:
   "DB1_SalidasExterioresDeMesa".Mesa[#Mesa].Ir_Pos_E2E4 := (#T1_ET60 OR #T1_ET20 OR #T1_ET21 OR (#T1_ET02 AND (#O_Sal_S4 OR ((#O_Bloqueo OR #O_Vaciar) AND #Mx_FlujoPrin_S4)))) AND NOT #PosTR_E2 AND #EstadoZona.Marcha_CBx AND NOT #EstadoVI.Error_Mx AND NOT #EstadoZona.Manual_CBx;
END_REGION

REGION Network 60: #MA_IR_POS_13_T
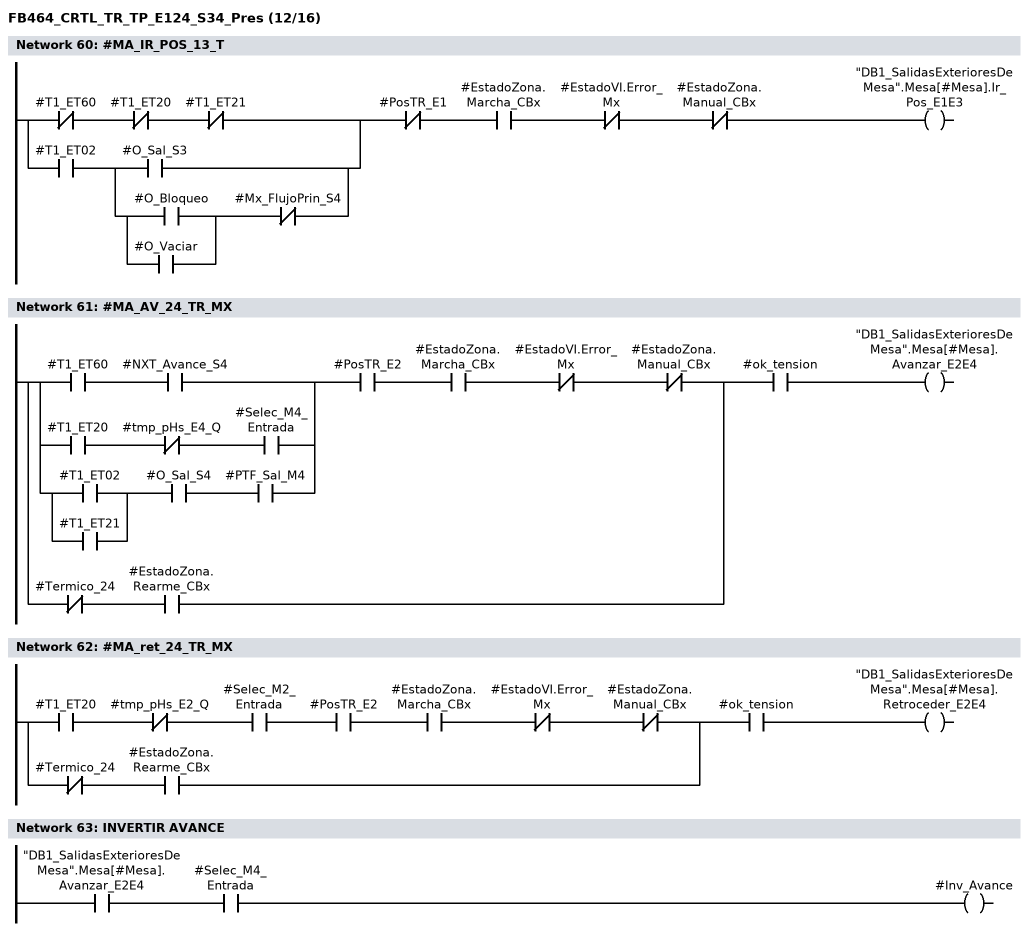
   RUNG wire#powerrail
      I_Contact( #T1_ET60 )
      I_Contact( #T1_ET20 )
      I_Contact( #T1_ET21 )
      wire#w1
      I_Contact( #PosTR_E1 )
      Contact( #EstadoZona.Marcha_CBx )
      I_Contact( #EstadoVI.Error_Mx )
      I_Contact( #EstadoZona.Manual_CBx )
      Coil( "DB1_SalidasExterioresDeMesa".Mesa[#Mesa].Ir_Pos_E1E3 )
   END_RUNG
   RUNG wire#powerrail
      Contact( #T1_ET02 )
      wire#w2
      Contact( #O_Sal_S3 )
   END_RUNG wire#w1
   RUNG wire#w2
      Contact( #O_Bloqueo )
      wire#w3
      I_Contact( #Mx_FlujoPrin_S4 )
   END_RUNG wire#w1
   RUNG wire#w2
      Contact( #O_Vaciar )
   END_RUNG wire#w3
   // the same network as SCL:
   "DB1_SalidasExterioresDeMesa".Mesa[#Mesa].Ir_Pos_E1E3 := ((NOT #T1_ET60 AND NOT #T1_ET20 AND NOT #T1_ET21) OR (#T1_ET02 AND (#O_Sal_S3 OR ((#O_Bloqueo OR #O_Vaciar) AND NOT #Mx_FlujoPrin_S4)))) AND NOT #PosTR_E1 AND #EstadoZona.Marcha_CBx AND NOT #EstadoVI.Error_Mx AND NOT #EstadoZona.Manual_CBx;
END_REGION

REGION Network 61: #MA_AV_24_TR_MX
   RUNG wire#powerrail
      Contact( #T1_ET60 )
      Contact( #NXT_Avance_S4 )
      wire#w1
      Contact( #PosTR_E2 )
      Contact( #EstadoZona.Marcha_CBx )
      I_Contact( #EstadoVI.Error_Mx )
      I_Contact( #EstadoZona.Manual_CBx )
      wire#w3
      Contact( #ok_tension )
      Coil( "DB1_SalidasExterioresDeMesa".Mesa[#Mesa].Avanzar_E2E4 )
   END_RUNG
   RUNG wire#powerrail
      Contact( #T1_ET20 )
      I_Contact( #tmp_pHs_E4_Q )
      Contact( #Selec_M4_Entrada )
   END_RUNG wire#w1
   RUNG wire#powerrail
      Contact( #T1_ET02 )
      wire#w2
      Contact( #O_Sal_S4 )
      Contact( #PTF_Sal_M4 )
   END_RUNG wire#w1
   RUNG wire#powerrail
      Contact( #T1_ET21 )
   END_RUNG wire#w2
   RUNG wire#powerrail
      I_Contact( #Termico_24 )
      Contact( #EstadoZona.Rearme_CBx )
   END_RUNG wire#w3
   // the same network as SCL:
   "DB1_SalidasExterioresDeMesa".Mesa[#Mesa].Avanzar_E2E4 := ((((#T1_ET60 AND #NXT_Avance_S4) OR (#T1_ET20 AND NOT #tmp_pHs_E4_Q AND #Selec_M4_Entrada) OR ((#T1_ET02 OR #T1_ET21) AND #O_Sal_S4 AND #PTF_Sal_M4)) AND #PosTR_E2 AND #EstadoZona.Marcha_CBx AND NOT #EstadoVI.Error_Mx AND NOT #EstadoZona.Manual_CBx) OR (NOT #Termico_24 AND #EstadoZona.Rearme_CBx)) AND #ok_tension;
END_REGION

REGION Network 62: #MA_ret_24_TR_MX
   RUNG wire#powerrail
      Contact( #T1_ET20 )
      I_Contact( #tmp_pHs_E2_Q )
      Contact( #Selec_M2_Entrada )
      Contact( #PosTR_E2 )
      Contact( #EstadoZona.Marcha_CBx )
      I_Contact( #EstadoVI.Error_Mx )
      I_Contact( #EstadoZona.Manual_CBx )
      wire#w1
      Contact( #ok_tension )
      Coil( "DB1_SalidasExterioresDeMesa".Mesa[#Mesa].Retroceder_E2E4 )
   END_RUNG
   RUNG wire#powerrail
      I_Contact( #Termico_24 )
      Contact( #EstadoZona.Rearme_CBx )
   END_RUNG wire#w1
   // the same network as SCL:
   "DB1_SalidasExterioresDeMesa".Mesa[#Mesa].Retroceder_E2E4 := ((#T1_ET20 AND NOT #tmp_pHs_E2_Q AND #Selec_M2_Entrada AND #PosTR_E2 AND #EstadoZona.Marcha_CBx AND NOT #EstadoVI.Error_Mx AND NOT #EstadoZona.Manual_CBx) OR (NOT #Termico_24 AND #EstadoZona.Rearme_CBx)) AND #ok_tension;
END_REGION

REGION Network 63: INVERTIR AVANCE
   RUNG wire#powerrail
      Contact( "DB1_SalidasExterioresDeMesa".Mesa[#Mesa].Avanzar_E2E4 )
      Contact( #Selec_M4_Entrada )
      Coil( #Inv_Avance )
   END_RUNG
   // the same network as SCL:
   #Inv_Avance := "DB1_SalidasExterioresDeMesa".Mesa[#Mesa].Avanzar_E2E4 AND #Selec_M4_Entrada;
END_REGION

REGION Network 64: #MA_AV_13_T_MX
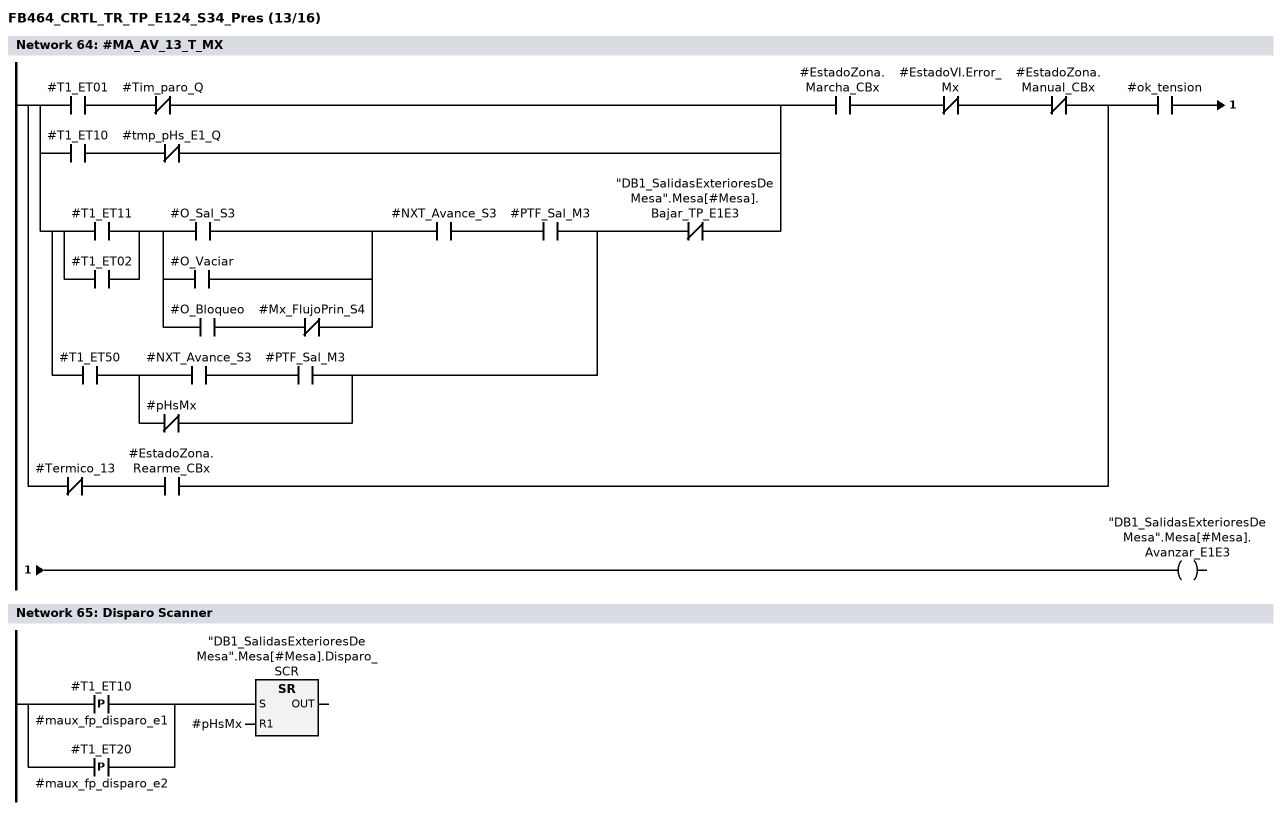
   RUNG wire#powerrail
      Contact( #T1_ET01 )
      I_Contact( #Tim_paro_Q )
      wire#w1
      Contact( #EstadoZona.Marcha_CBx )
      I_Contact( #EstadoVI.Error_Mx )
      I_Contact( #EstadoZona.Manual_CBx )
      wire#w6
      Contact( #ok_tension )
      Coil( "DB1_SalidasExterioresDeMesa".Mesa[#Mesa].Avanzar_E1E3 )
   END_RUNG
   RUNG wire#powerrail
      Contact( #T1_ET10 )
      I_Contact( #tmp_pHs_E1_Q )
   END_RUNG wire#w1
   RUNG wire#powerrail
      Contact( #T1_ET11 )
      wire#w2
      Contact( #O_Sal_S3 )
      wire#w3
      Contact( #NXT_Avance_S3 )
      Contact( #PTF_Sal_M3 )
      wire#w4
      I_Contact( "DB1_SalidasExterioresDeMesa".Mesa[#Mesa].Bajar_TP_E1E3 )
   END_RUNG wire#w1
   RUNG wire#powerrail
      Contact( #T1_ET02 )
   END_RUNG wire#w2
   RUNG wire#w2
      Contact( #O_Vaciar )
   END_RUNG wire#w3
   RUNG wire#w2
      Contact( #O_Bloqueo )
      I_Contact( #Mx_FlujoPrin_S4 )
   END_RUNG wire#w3
   RUNG wire#powerrail
      Contact( #T1_ET50 )
      wire#w5
      Contact( #NXT_Avance_S3 )
      Contact( #PTF_Sal_M3 )
   END_RUNG wire#w4
   RUNG wire#w5
      I_Contact( #pHsMx )
   END_RUNG wire#w4
   RUNG wire#powerrail
      I_Contact( #Termico_13 )
      Contact( #EstadoZona.Rearme_CBx )
   END_RUNG wire#w6
   // the same network as SCL:
   "DB1_SalidasExterioresDeMesa".Mesa[#Mesa].Avanzar_E1E3 := ((((#T1_ET01 AND NOT #Tim_paro_Q) OR (#T1_ET10 AND NOT #tmp_pHs_E1_Q) OR ((((#T1_ET11 OR #T1_ET02) AND (#O_Sal_S3 OR #O_Vaciar OR (#O_Bloqueo AND NOT #Mx_FlujoPrin_S4)) AND #NXT_Avance_S3 AND #PTF_Sal_M3) OR (#T1_ET50 AND ((#NXT_Avance_S3 AND #PTF_Sal_M3) OR NOT #pHsMx))) AND NOT "DB1_SalidasExterioresDeMesa".Mesa[#Mesa].Bajar_TP_E1E3)) AND #EstadoZona.Marcha_CBx AND NOT #EstadoVI.Error_Mx AND NOT #EstadoZona.Manual_CBx) OR (NOT #Termico_13 AND #EstadoZona.Rearme_CBx)) AND #ok_tension;
END_REGION

REGION Network 65: Disparo Scanner
   RUNG wire#powerrail
      P_Contact(operand := #T1_ET10, bit := #maux_fp_disparo_e1)
      wire#w1
      S_SR(operand := "DB1_SalidasExterioresDeMesa".Mesa[#Mesa].Disparo_SCR, r1 := #pHsMx)
   END_RUNG
   RUNG wire#powerrail
      P_Contact(operand := #T1_ET20, bit := #maux_fp_disparo_e2)
   END_RUNG wire#w1
   // the same network as SCL:
   #_w1 := #T1_ET10 AND NOT #maux_fp_disparo_e1;   // rising edge of #T1_ET10
   #maux_fp_disparo_e1 := #T1_ET10;
   #_w2 := #T1_ET20 AND NOT #maux_fp_disparo_e2;   // rising edge of #T1_ET20
   #maux_fp_disparo_e2 := #T1_ET20;
   IF #_w1 OR #_w2 THEN
       "DB1_SalidasExterioresDeMesa".Mesa[#Mesa].Disparo_SCR := TRUE;   // SR flip-flop
   END_IF;
   IF #pHsMx THEN "DB1_SalidasExterioresDeMesa".Mesa[#Mesa].Disparo_SCR := FALSE; END_IF;
END_REGION

REGION Network 66: PASAR ETIQUETA JDT
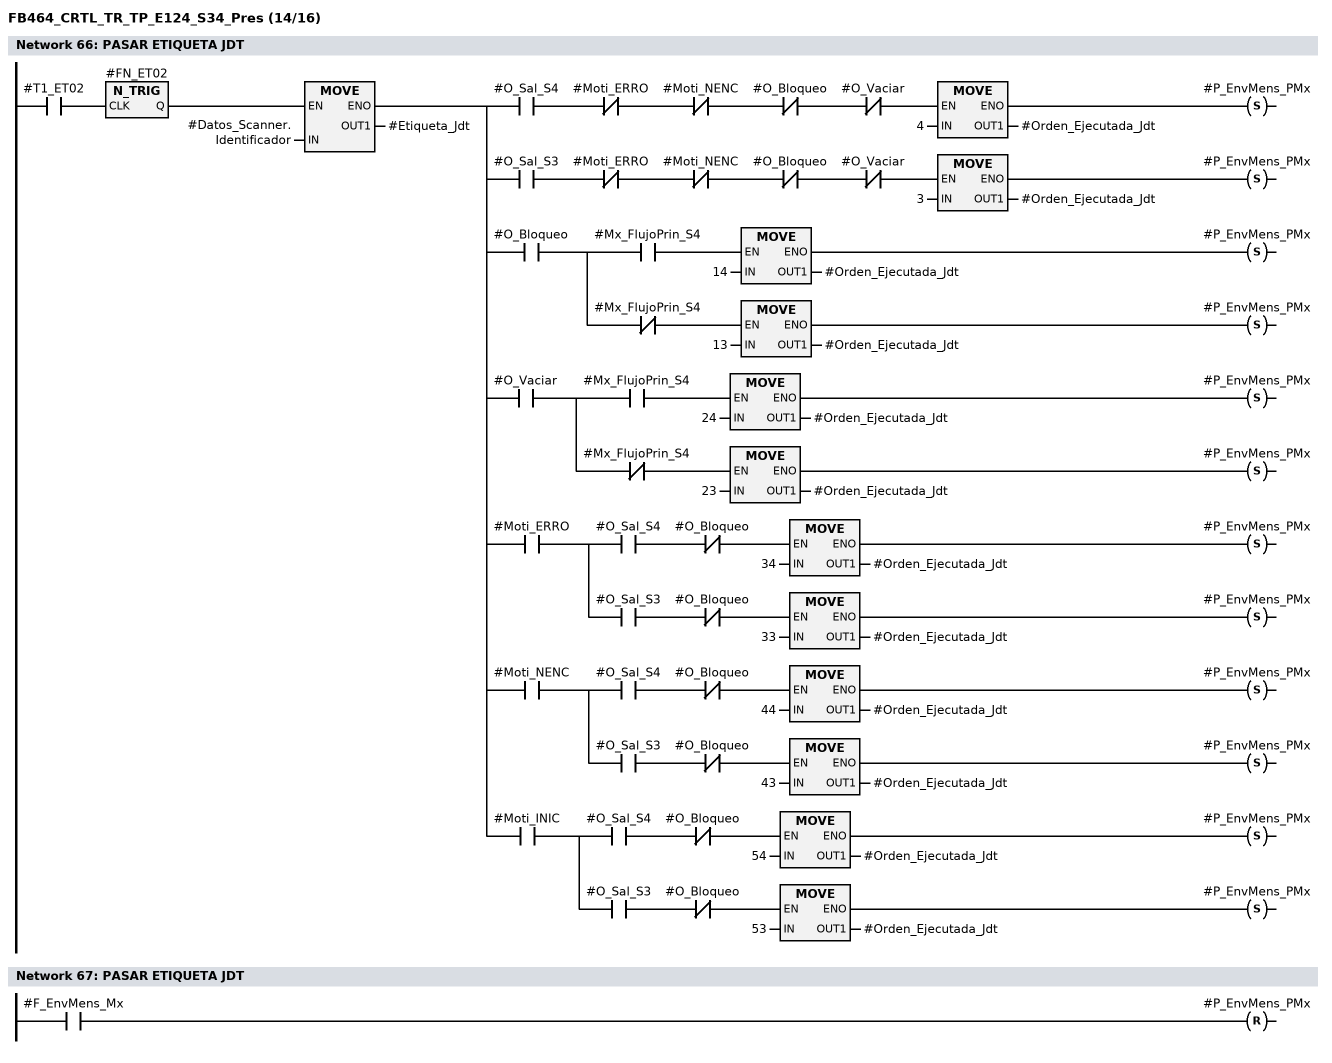
   RUNG wire#powerrail
      Contact( #T1_ET02 )
      N_Trig( #FN_ET02 )
      { S7_GenerateENO := "TRUE" } Move(in := #Datos_Scanner.Identificador, out1 => #Etiqueta_Jdt)
      wire#w1
      Contact( #O_Sal_S4 )
      I_Contact( #Moti_ERRO )
      I_Contact( #Moti_NENC )
      I_Contact( #O_Bloqueo )
      I_Contact( #O_Vaciar )
      { S7_GenerateENO := "TRUE" } Move(in := 4, out1 => #Orden_Ejecutada_Jdt)
      S_Coil( #P_EnvMens_PMx )
   END_RUNG
   RUNG wire#w1
      Contact( #O_Sal_S3 )
      I_Contact( #Moti_ERRO )
      I_Contact( #Moti_NENC )
      I_Contact( #O_Bloqueo )
      I_Contact( #O_Vaciar )
      { S7_GenerateENO := "TRUE" } Move(in := 3, out1 => #Orden_Ejecutada_Jdt)
      S_Coil( #P_EnvMens_PMx )
   END_RUNG
   RUNG wire#w1
      Contact( #O_Bloqueo )
      wire#w2
      Contact( #Mx_FlujoPrin_S4 )
      { S7_GenerateENO := "TRUE" } Move(in := 14, out1 => #Orden_Ejecutada_Jdt)
      S_Coil( #P_EnvMens_PMx )
   END_RUNG
   RUNG wire#w2
      I_Contact( #Mx_FlujoPrin_S4 )
      { S7_GenerateENO := "TRUE" } Move(in := 13, out1 => #Orden_Ejecutada_Jdt)
      S_Coil( #P_EnvMens_PMx )
   END_RUNG
   RUNG wire#w1
      Contact( #O_Vaciar )
      wire#w3
      Contact( #Mx_FlujoPrin_S4 )
      { S7_GenerateENO := "TRUE" } Move(in := 24, out1 => #Orden_Ejecutada_Jdt)
      S_Coil( #P_EnvMens_PMx )
   END_RUNG
   RUNG wire#w3
      I_Contact( #Mx_FlujoPrin_S4 )
      { S7_GenerateENO := "TRUE" } Move(in := 23, out1 => #Orden_Ejecutada_Jdt)
      S_Coil( #P_EnvMens_PMx )
   END_RUNG
   RUNG wire#w1
      Contact( #Moti_ERRO )
      wire#w4
      Contact( #O_Sal_S4 )
      I_Contact( #O_Bloqueo )
      { S7_GenerateENO := "TRUE" } Move(in := 34, out1 => #Orden_Ejecutada_Jdt)
      S_Coil( #P_EnvMens_PMx )
   END_RUNG
   RUNG wire#w4
      Contact( #O_Sal_S3 )
      I_Contact( #O_Bloqueo )
      { S7_GenerateENO := "TRUE" } Move(in := 33, out1 => #Orden_Ejecutada_Jdt)
      S_Coil( #P_EnvMens_PMx )
   END_RUNG
   RUNG wire#w1
      Contact( #Moti_NENC )
      wire#w5
      Contact( #O_Sal_S4 )
      I_Contact( #O_Bloqueo )
      { S7_GenerateENO := "TRUE" } Move(in := 44, out1 => #Orden_Ejecutada_Jdt)
      S_Coil( #P_EnvMens_PMx )
   END_RUNG
   RUNG wire#w5
      Contact( #O_Sal_S3 )
      I_Contact( #O_Bloqueo )
      { S7_GenerateENO := "TRUE" } Move(in := 43, out1 => #Orden_Ejecutada_Jdt)
      S_Coil( #P_EnvMens_PMx )
   END_RUNG
   RUNG wire#w1
      Contact( #Moti_INIC )
      wire#w6
      Contact( #O_Sal_S4 )
      I_Contact( #O_Bloqueo )
      { S7_GenerateENO := "TRUE" } Move(in := 54, out1 => #Orden_Ejecutada_Jdt)
      S_Coil( #P_EnvMens_PMx )
   END_RUNG
   RUNG wire#w6
      Contact( #O_Sal_S3 )
      I_Contact( #O_Bloqueo )
      { S7_GenerateENO := "TRUE" } Move(in := 53, out1 => #Orden_Ejecutada_Jdt)
      S_Coil( #P_EnvMens_PMx )
   END_RUNG
   // the same network as SCL:
   // ENO of a box is taken as its EN; it also drops when the box reports an error
   #_w1 := NOT #T1_ET02 AND #FN_ET02;   // falling edge
   #FN_ET02 := #T1_ET02;
   IF #_w1 THEN #Etiqueta_Jdt := #Datos_Scanner.Identificador; END_IF;
   IF #_w1 AND #O_Sal_S4 AND NOT #Moti_ERRO AND NOT #Moti_NENC AND NOT #O_Bloqueo AND NOT #O_Vaciar THEN
       #Orden_Ejecutada_Jdt := 4;
       #P_EnvMens_PMx := TRUE;
   END_IF;
   IF #_w1 AND #O_Sal_S3 AND NOT #Moti_ERRO AND NOT #Moti_NENC AND NOT #O_Bloqueo AND NOT #O_Vaciar THEN
       #Orden_Ejecutada_Jdt := 3;
       #P_EnvMens_PMx := TRUE;
   END_IF;
   #_w2 := #_w1 AND #O_Bloqueo;
   IF #_w2 AND #Mx_FlujoPrin_S4 THEN
       #Orden_Ejecutada_Jdt := 14;
       #P_EnvMens_PMx := TRUE;
   END_IF;
   IF #_w2 AND NOT #Mx_FlujoPrin_S4 THEN
       #Orden_Ejecutada_Jdt := 13;
       #P_EnvMens_PMx := TRUE;
   END_IF;
   #_w3 := #_w1 AND #O_Vaciar;
   IF #_w3 AND #Mx_FlujoPrin_S4 THEN
       #Orden_Ejecutada_Jdt := 24;
       #P_EnvMens_PMx := TRUE;
   END_IF;
   IF #_w3 AND NOT #Mx_FlujoPrin_S4 THEN
       #Orden_Ejecutada_Jdt := 23;
       #P_EnvMens_PMx := TRUE;
   END_IF;
   #_w4 := #_w1 AND #Moti_ERRO;
   IF #_w4 AND #O_Sal_S4 AND NOT #O_Bloqueo THEN
       #Orden_Ejecutada_Jdt := 34;
       #P_EnvMens_PMx := TRUE;
   END_IF;
   IF #_w4 AND #O_Sal_S3 AND NOT #O_Bloqueo THEN
       #Orden_Ejecutada_Jdt := 33;
       #P_EnvMens_PMx := TRUE;
   END_IF;
   #_w5 := #_w1 AND #Moti_NENC;
   IF #_w5 AND #O_Sal_S4 AND NOT #O_Bloqueo THEN
       #Orden_Ejecutada_Jdt := 44;
       #P_EnvMens_PMx := TRUE;
   END_IF;
   IF #_w5 AND #O_Sal_S3 AND NOT #O_Bloqueo THEN
       #Orden_Ejecutada_Jdt := 43;
       #P_EnvMens_PMx := TRUE;
   END_IF;
   #_w6 := #_w1 AND #Moti_INIC;
   IF #_w6 AND #O_Sal_S4 AND NOT #O_Bloqueo THEN
       #Orden_Ejecutada_Jdt := 54;
       #P_EnvMens_PMx := TRUE;
   END_IF;
   IF #_w6 AND #O_Sal_S3 AND NOT #O_Bloqueo THEN
       #Orden_Ejecutada_Jdt := 53;
       #P_EnvMens_PMx := TRUE;
   END_IF;
END_REGION

REGION Network 67: PASAR ETIQUETA JDT
   RUNG wire#powerrail
      Contact( #F_EnvMens_Mx )
      R_Coil( #P_EnvMens_PMx )
   END_RUNG
   // the same network as SCL:
   IF #F_EnvMens_Mx THEN #P_EnvMens_PMx := FALSE; END_IF;
END_REGION

REGION Network 68: ESTADOS MESA
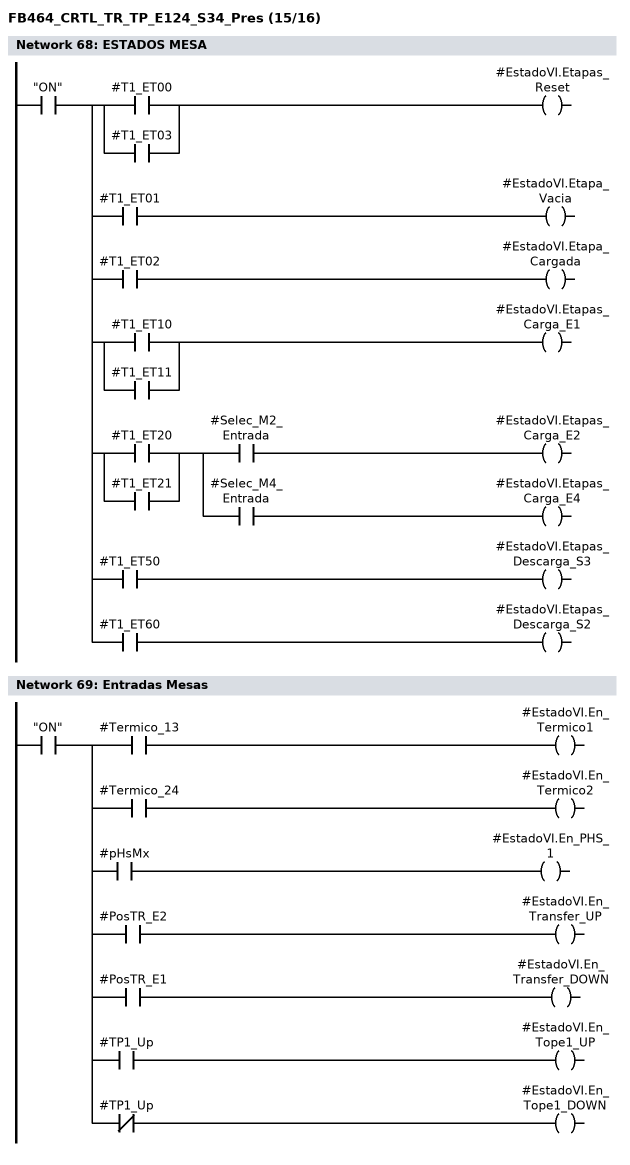
   RUNG wire#powerrail
      Contact( "ON" )
      wire#w1
      Contact( #T1_ET00 )
      wire#w2
      Coil( #EstadoVI.Etapas_Reset )
   END_RUNG
   RUNG wire#w1
      Contact( #T1_ET03 )
   END_RUNG wire#w2
   RUNG wire#w1
      Contact( #T1_ET01 )
      Coil( #EstadoVI.Etapa_Vacia )
   END_RUNG
   RUNG wire#w1
      Contact( #T1_ET02 )
      Coil( #EstadoVI.Etapa_Cargada )
   END_RUNG
   RUNG wire#w1
      Contact( #T1_ET10 )
      wire#w3
      Coil( #EstadoVI.Etapas_Carga_E1 )
   END_RUNG
   RUNG wire#w1
      Contact( #T1_ET11 )
   END_RUNG wire#w3
   RUNG wire#w1
      Contact( #T1_ET20 )
      wire#w4
      Contact( #Selec_M2_Entrada )
      Coil( #EstadoVI.Etapas_Carga_E2 )
   END_RUNG
   RUNG wire#w1
      Contact( #T1_ET21 )
   END_RUNG wire#w4
   RUNG wire#w4
      Contact( #Selec_M4_Entrada )
      Coil( #EstadoVI.Etapas_Carga_E4 )
   END_RUNG
   RUNG wire#w1
      Contact( #T1_ET50 )
      Coil( #EstadoVI.Etapas_Descarga_S3 )
   END_RUNG
   RUNG wire#w1
      Contact( #T1_ET60 )
      Coil( #EstadoVI.Etapas_Descarga_S2 )
   END_RUNG
   // the same network as SCL:
   #EstadoVI.Etapas_Reset := "ON" AND (#T1_ET00 OR #T1_ET03);
   #EstadoVI.Etapa_Vacia := "ON" AND #T1_ET01;
   #EstadoVI.Etapa_Cargada := "ON" AND #T1_ET02;
   #EstadoVI.Etapas_Carga_E1 := "ON" AND (#T1_ET10 OR #T1_ET11);
   #_w1 := "ON" AND (#T1_ET20 OR #T1_ET21);
   #EstadoVI.Etapas_Carga_E2 := #_w1 AND #Selec_M2_Entrada;
   #EstadoVI.Etapas_Carga_E4 := #_w1 AND #Selec_M4_Entrada;
   #EstadoVI.Etapas_Descarga_S3 := "ON" AND #T1_ET50;
   #EstadoVI.Etapas_Descarga_S2 := "ON" AND #T1_ET60;
END_REGION

REGION Network 69: Entradas Mesas
   RUNG wire#powerrail
      Contact( "ON" )
      wire#w1
      Contact( #Termico_13 )
      Coil( #EstadoVI.En_Termico1 )
   END_RUNG
   RUNG wire#w1
      Contact( #Termico_24 )
      Coil( #EstadoVI.En_Termico2 )
   END_RUNG
   RUNG wire#w1
      Contact( #pHsMx )
      Coil( #EstadoVI.En_PHS_1 )
   END_RUNG
   RUNG wire#w1
      Contact( #PosTR_E2 )
      Coil( #EstadoVI.En_Transfer_UP )
   END_RUNG
   RUNG wire#w1
      Contact( #PosTR_E1 )
      Coil( #EstadoVI.En_Transfer_DOWN )
   END_RUNG
   RUNG wire#w1
      Contact( #TP1_Up )
      Coil( #EstadoVI.En_Tope1_UP )
   END_RUNG
   RUNG wire#w1
      I_Contact( #TP1_Up )
      Coil( #EstadoVI.En_Tope1_DOWN )
   END_RUNG
   // the same network as SCL:
   #EstadoVI.En_Termico1 := "ON" AND #Termico_13;
   #EstadoVI.En_Termico2 := "ON" AND #Termico_24;
   #EstadoVI.En_PHS_1 := "ON" AND #pHsMx;
   #EstadoVI.En_Transfer_UP := "ON" AND #PosTR_E2;
   #EstadoVI.En_Transfer_DOWN := "ON" AND #PosTR_E1;
   #EstadoVI.En_Tope1_UP := "ON" AND #TP1_Up;
   #EstadoVI.En_Tope1_DOWN := "ON" AND NOT #TP1_Up;
END_REGION

REGION Network 70: Salidas Mesas
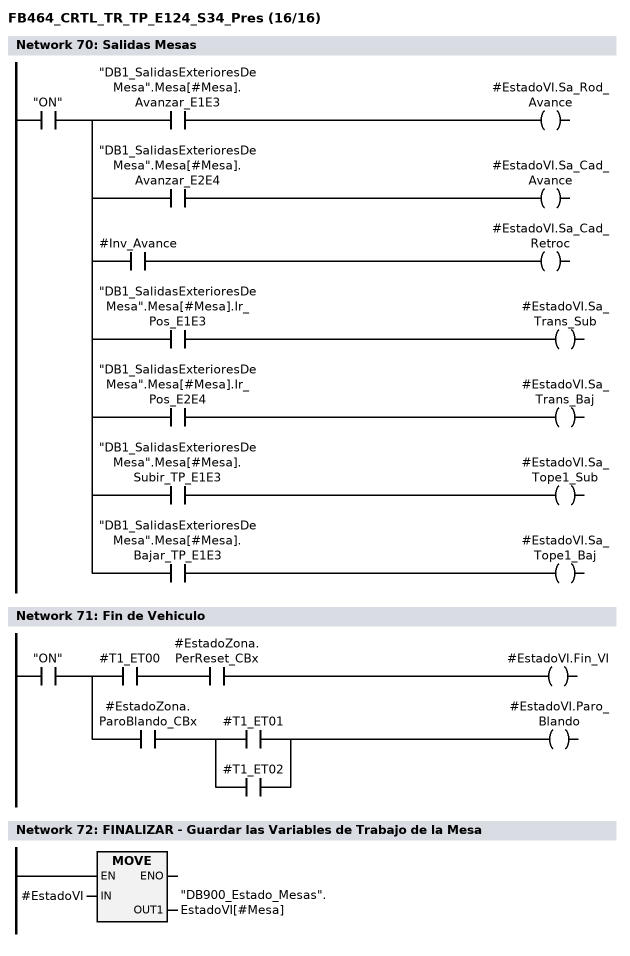
   RUNG wire#powerrail
      Contact( "ON" )
      wire#w1
      Contact( "DB1_SalidasExterioresDeMesa".Mesa[#Mesa].Avanzar_E1E3 )
      Coil( #EstadoVI.Sa_Rod_Avance )
   END_RUNG
   RUNG wire#w1
      Contact( "DB1_SalidasExterioresDeMesa".Mesa[#Mesa].Avanzar_E2E4 )
      Coil( #EstadoVI.Sa_Cad_Avance )
   END_RUNG
   RUNG wire#w1
      Contact( #Inv_Avance )
      Coil( #EstadoVI.Sa_Cad_Retroc )
   END_RUNG
   RUNG wire#w1
      Contact( "DB1_SalidasExterioresDeMesa".Mesa[#Mesa].Ir_Pos_E1E3 )
      Coil( #EstadoVI.Sa_Trans_Sub )
   END_RUNG
   RUNG wire#w1
      Contact( "DB1_SalidasExterioresDeMesa".Mesa[#Mesa].Ir_Pos_E2E4 )
      Coil( #EstadoVI.Sa_Trans_Baj )
   END_RUNG
   RUNG wire#w1
      Contact( "DB1_SalidasExterioresDeMesa".Mesa[#Mesa].Subir_TP_E1E3 )
      Coil( #EstadoVI.Sa_Tope1_Sub )
   END_RUNG
   RUNG wire#w1
      Contact( "DB1_SalidasExterioresDeMesa".Mesa[#Mesa].Bajar_TP_E1E3 )
      Coil( #EstadoVI.Sa_Tope1_Baj )
   END_RUNG
   // the same network as SCL:
   #EstadoVI.Sa_Rod_Avance := "ON" AND "DB1_SalidasExterioresDeMesa".Mesa[#Mesa].Avanzar_E1E3;
   #EstadoVI.Sa_Cad_Avance := "ON" AND "DB1_SalidasExterioresDeMesa".Mesa[#Mesa].Avanzar_E2E4;
   #EstadoVI.Sa_Cad_Retroc := "ON" AND #Inv_Avance;
   #EstadoVI.Sa_Trans_Sub := "ON" AND "DB1_SalidasExterioresDeMesa".Mesa[#Mesa].Ir_Pos_E1E3;
   #EstadoVI.Sa_Trans_Baj := "ON" AND "DB1_SalidasExterioresDeMesa".Mesa[#Mesa].Ir_Pos_E2E4;
   #EstadoVI.Sa_Tope1_Sub := "ON" AND "DB1_SalidasExterioresDeMesa".Mesa[#Mesa].Subir_TP_E1E3;
   #EstadoVI.Sa_Tope1_Baj := "ON" AND "DB1_SalidasExterioresDeMesa".Mesa[#Mesa].Bajar_TP_E1E3;
END_REGION

REGION Network 71: Fin de Vehiculo
   RUNG wire#powerrail
      Contact( "ON" )
      wire#w1
      Contact( #T1_ET00 )
      Contact( #EstadoZona.PerReset_CBx )
      Coil( #EstadoVI.Fin_VI )
   END_RUNG
   RUNG wire#w1
      Contact( #EstadoZona.ParoBlando_CBx )
      wire#w2
      Contact( #T1_ET01 )
      wire#w3
      Coil( #EstadoVI.Paro_Blando )
   END_RUNG
   RUNG wire#w2
      Contact( #T1_ET02 )
   END_RUNG wire#w3
   // the same network as SCL:
   #EstadoVI.Fin_VI := "ON" AND #T1_ET00 AND #EstadoZona.PerReset_CBx;
   #EstadoVI.Paro_Blando := "ON" AND #EstadoZona.ParoBlando_CBx AND (#T1_ET01 OR #T1_ET02);
END_REGION

REGION Network 72: FINALIZAR - Guardar las Variables de Trabajo de la Mesa
   RUNG wire#powerrail
      Move(in := #EstadoVI, out1 => "DB900_Estado_Mesas".EstadoVI[#Mesa])
   END_RUNG
   // the same network as SCL:
   "DB900_Estado_Mesas".EstadoVI[#Mesa] := #EstadoVI;
END_REGION
END_FUNCTION_BLOCK
